	saAux[0] := ('UPDATE `geral`.`processos` SET `InicioAspersao` = $'');
	saAux[1] := (TO_STRING(camara.en.stHoraAgora.wYear));
	saAux[2] := ('-');
	saAux[3] := (TO_STRING(camara.en.stHoraAgora.wMonth));
	saAux[4] := ('-');
	saAux[5] := (TO_STRING(camara.en.stHoraAgora.wDay));
	saAux[6] := (' ');
	saAux[7] := (TO_STRING(camara.en.stHoraAgora.wHour));
	saAux[8] := (':');
	saAux[9] := (TO_STRING(camara.en.stHoraAgora.wMinute));
	saAux[10] := (':');
	saAux[11] := (TO_STRING(camara.en.stHoraAgora.wSecond));
	saAux[12] := ('$' WHERE (`Processo` = $'');
	saAux[13] := (sGuidAnterior);
	saAux[14] := ('$');');
	
	sCmd := F_ConcatArray1000(sArray:= saAux);
	
	aPara.eParaType := E_ExpParameterType.STRING_;
	aPara.nParaSize := SIZEOF(sAux);

	// call functionblock
	IF fbPLCDBaspersao.Execute(
		hDBID:= 1, 
		pExpression:= ADR(sCmd), 
		cbExpression:= SIZEOF(sCmd), 
		pData:= ADR(sAux), 
		cbData:= SIZEOF(sAux), 
		pParameter:= ADR(aPara), 
		cbParameter:= SIZEOF(aPara)) 
	THEN
		IF NOT fbPLCDBaspersao.bError THEN
			xSalvaInicioAspersao := FALSE;
		END_IF
	END_IF
END_IF
END_ACTION

ACTION InicioResfriamento:



//UPDATE `geral`.`processos` SET `InicioResfriamento` = '1', `NumeroCarcacas` = '1' WHERE (`Processo` = '{F4C353B8-2323-45D1-B9F0-8A1F447BE435}');


IF xSalvaResfriamento THEN
	
	FOR i:= 0 TO 50 DO
		saAux[i]:= '';
	END_FOR
	
	saAux[0] := ('UPDATE `geral`.`processos` SET `InicioResfriamento` = $'');
	saAux[2] := (TO_STRING(camara.en.stHoraAgora.wYear));
	saAux[3] := ('-');
	saAux[4] := (TO_STRING(camara.en.stHoraAgora.wMonth));
	saAux[5] := ('-');
	saAux[6] := (TO_STRING(camara.en.stHoraAgora.wDay));
	saAux[7] := (' ');
	saAux[8] := (TO_STRING(camara.en.stHoraAgora.wHour));
	saAux[9] := (':');
	saAux[10] := (TO_STRING(camara.en.stHoraAgora.wMinute));
	saAux[11] := (':');
	saAux[12] := (TO_STRING(stHoraAhora.wSecond));
	saAux[13] := ('$', `NumeroCarcacas` = $'');
	saAux[14] := (TO_STRING(Camara.config.iCarcacasReal));
	saAux[15] := ('$', `Camara` = $'');
	saAux[16] := (TO_STRING(Camara.config.iCamara));
	saAux[17] := ('$' WHERE (`Processo` = $'');
	saAux[18] := (sGuidAnterior);
	saAux[19] := ('$');');
	
	sCmd := F_ConcatArray1000(sArray:= saAux);
	
	aPara.eParaType := E_ExpParameterType.STRING_;
	aPara.nParaSize := SIZEOF(sAux);

	// call functionblock
	IF fbPLCDBResfriamento.Execute(
		hDBID:= 1, 
		pExpression:= ADR(sCmd), 
		cbExpression:= SIZEOF(sCmd), 
		pData:= ADR(sAux), 
		cbData:= SIZEOF(sAux), 
		pParameter:= ADR(aPara), 
		cbParameter:= SIZEOF(aPara)) 
	THEN
		IF NOT fbPLCDBResfriamento.bError THEN
			xSalvaResfriamento := FALSE;
		END_IF
	END_IF
END_IF
END_ACTION

ACTION SalvaGrafico:



//INSERT INTO `geral`.`graficosprocesso` (`Processo`, `rTempTanque`, `rPressaoAnel`, `rUmidadeCamara`, `timestamp`) VALUES ('s', 's', 's', 's', 's');

tonAmostra(IN:= sGuidAtual <> '' AND xAmostra, PT:= T#1M, Q=> , ET=> );
IF tonAmostra.q THEN
	tonAmostra(IN:= FALSE);
	xSalvaGrafico := TRUE;
END_IF


IF xSalvaGrafico THEN
	
	FOR i:= 0 TO 50 DO
		saAux[i]:= '';
	END_FOR
	
	
	saAux[0]:= ('INSERT INTO `geral`.`graficoscamara` (`Processo`, `rUmidadeCamara`, `rTem');
	saAux[1]:= ('peraturaCamara`,`rVazaoCamara`,`rPressaoAnel`,`rTempReservatorio`');
	saAux[2]:= (', `timestamp`) VALUES ($'');
	saAux[3]:= (sGuidAnterior);
	saAux[4]:= ('$', $'');
	saAux[5]:= (TO_STRING(F_RetiraCasa(Entrada:= Camara.en.rUmidadeCamara, casa:=2)));
	saAux[6]:= ('$', $'');
	saAux[7]:= (TO_STRING(F_RetiraCasa(Entrada:= Camara.en.rTempCamara, casa:=2)));
	saAux[8]:= ('$', $'');
	saAux[9]:= (TO_STRING(F_RetiraCasa(Entrada:= Camara.en.rVaozaoInstantanea, casa:=2)));
	saAux[10]:= ('$', $'');
	saAux[11]:= (TO_STRING(F_RetiraCasa(Entrada:= Camara.en.rPressaoAnel, casa:=2)));
	saAux[12]:= ('$', $'');
	saAux[13]:= (TO_STRING(F_RetiraCasa(Entrada:= Camara.en.rTempTanque, casa:=2)));
	saAux[14]:= ('$', $'');
	saAux[15]:= (TO_STRING(camara.en.stHoraAgora.wYear));
	saAux[16]:= ('-');
	saAux[17]:= (TO_STRING(camara.en.stHoraAgora.wMonth));
	saAux[18]:= ('-');
	saAux[19]:= (TO_STRING(camara.en.stHoraAgora.wDay));
	saAux[20]:= (' ');
	saAux[21]:= (TO_STRING(camara.en.stHoraAgora.wHour));
	saAux[22]:= (':');
	saAux[23]:= (TO_STRING(camara.en.stHoraAgora.wMinute));
	saAux[24]:= (':');
	saAux[25]:= (TO_STRING(camara.en.stHoraAgora.wSecond));
	saAux[26]:= ('$');');
	
	sCmd := F_ConcatArray1000(sArray:= saAux);
	
	aPara.eParaType := E_ExpParameterType.STRING_;
	aPara.nParaSize := SIZEOF(sAux);

	// call functionblock
	IF fbPLCDBCmd.Execute(
		hDBID:= 1, 
		pExpression:= ADR(sCmd), 
		cbExpression:= SIZEOF(sCmd), 
		pData:= ADR(sAux), 
		cbData:= SIZEOF(sAux), 
		pParameter:= ADR(aPara), 
		cbParameter:= SIZEOF(aPara)) 
	THEN
		xSalvaGrafico := FALSE;
	END_IF
END_IF
END_ACTION

ACTION SalvaProtocolo:

IF xSalvaProtocolo THEN
		
	FOR i:= 0 TO 50 DO
		saAux[i]:= '';
	END_FOR

	//UPDATE `geral`.`processos` SET `sProtocolo` = 'aaaaaaa' WHERE (`Processo` = '{008089BB-BE64-417E-ABDE-888FE5FB9663}');

	saAux[0] := ('UPDATE `geral`.`processos` SET `sProtocolo` = $'');
	saAux[1] := (Camara.config.stProtocolos[Camara.config.iProtocoloEscolhido].DB.Nome);
	saAux[2] := ('$' WHERE (`Processo` = $'');
	saAux[3] := (sGuidAnterior);
	saAux[4] := ('$');');
	
	sCmd := F_ConcatArray1000(sArray:= saAux);
	
	aPara.eParaType := E_ExpParameterType.STRING_;
	aPara.nParaSize := SIZEOF(sAux);

	// call functionblock
	IF fbPLCDProtocolo.Execute(
		hDBID:= 1, 
		pExpression:= ADR(sCmd), 
		cbExpression:= SIZEOF(sCmd), 
		pData:= ADR(sAux), 
		cbData:= SIZEOF(sAux), 
		pParameter:= ADR(aPara), 
		cbParameter:= SIZEOF(aPara)) 
	THEN
		IF NOT fbPLCDProtocolo.bError THEN
			xSalvaProtocolo := FALSE;
		END_IF
	END_IF
END_IF
END_ACTION

ACTION AjustaEntrada:



IF Camara.config.iCamara <> CamaraAnterior.config.iCamara THEN
	iCamara := Camara.config.iCamara;
END_IF
IF Camara.config.iCamara <> iCamara THEN
	Camara.config.iCamara := iCamara;
END_IF


IF Camara.config.sNome <> CamaraAnterior.config.sNome THEN
	sNome := Camara.config.sNome;
END_IF
IF Camara.config.sNome <> sNome THEN
	Camara.config.sNome := sNome;
END_IF


IF Camara.en.sGuidAtual <> CamaraAnterior.en.sGuidAtual THEN
	sGuidAtual := Camara.en.sGuidAtual;
END_IF
IF Camara.en.sGuidAtual <> sGuidAtual THEN
	Camara.en.sGuidAtual := sGuidAtual;
END_IF


IF Camara.config.sValvulas <> CamaraAnterior.config.sValvulas THEN
	sValvulas := Camara.config.sValvulas;
	F_StringSeparadorFBGrupos(sStr:= sValvulas, ListaINT:=iValvulas);
END_IF
IF Camara.config.sValvulas <> sValvulas THEN
	Camara.config.sValvulas := sValvulas;
	F_StringSeparadorFBGrupos(sStr:= sValvulas, ListaINT:=iValvulas);
END_IF


IF Camara.status.xCamaraTempOK <> CamaraAnterior.status.xCamaraTempOK THEN
	xCamaraTempOK := Camara.status.xCamaraTempOK;
END_IF
IF Camara.status.xCamaraTempOK <> xCamaraTempOK THEN
	Camara.status.xCamaraTempOK := xCamaraTempOK;
END_IF

IF Camara.status.xCamaraUmidOK <> CamaraAnterior.status.xCamaraUmidOK THEN
	xCamaraUmidOK := Camara.status.xCamaraUmidOK;
END_IF
IF Camara.status.xCamaraUmidOK <> xCamaraUmidOK THEN
	Camara.status.xCamaraUmidOK := xCamaraUmidOK;
END_IF

IF Camara.status.xAnelPressOK <> CamaraAnterior.status.xAnelPressOK THEN
	xAnelPressOK := Camara.status.xAnelPressOK;
END_IF
IF Camara.status.xAnelPressOK <> xAnelPressOK THEN
	Camara.status.xAnelPressOK := xAnelPressOK;
END_IF

IF Camara.status.xTanqueTempOK <> CamaraAnterior.status.xTanqueTempOK THEN
	xTanqueTempOK := Camara.status.xTanqueTempOK;
END_IF
IF Camara.status.xTanqueTempOK <> xTanqueTempOK THEN
	Camara.status.xTanqueTempOK := xTanqueTempOK;
END_IF

IF Camara.en.xFinalizaValvulasDaCamara <> CamaraAnterior.en.xFinalizaValvulasDaCamara THEN
	xFinalizaValvulasDaCamara := Camara.en.xFinalizaValvulasDaCamara;
END_IF
IF Camara.en.xFinalizaValvulasDaCamara <> xFinalizaValvulasDaCamara THEN
	Camara.en.xFinalizaValvulasDaCamara := xFinalizaValvulasDaCamara;
END_IF

//Quantidade minima de carcaças a amostrar
IF Camara.config.iCarcacasAmostra < 20 THEN
	Camara.config.iCarcacasAmostra := 20;
END_IF



CamaraAnterior := Camara;
END_ACTION

ACTION AjustaSaida:




Camara.status.sStatus := sStatus;
Camara.status.iStatus := iStatus;
Camara.status.xTerminouAspercao := xTerminouAspercao;
Camara.sa.iQuantidadeDeCluster := iQuantidadeDeCluster;

Camara.status.sNomeProtocoloAtivo := Camara.config.stProtocolos[Camara.sa.iProtocoloAtual].DB.Nome;



Camara.sa.iValvulaMestraMestra := iValvulaMestraMestra;
END_ACTION

ACTION BTPausaECancela:




//Sinal de cancela todas as valvulas
btCancela(CLK:= Camara.en.xCancelaTodas, Q=> );
IF btCancela.q THEN
	xIniciaCascataCancela := TRUE;
END_IF
tonCascataCancela(IN:= xIniciaCascataCancela, PT:= T#250MS, Q=> , ET=> );
IF tonCascataCancela.q THEN
	tonCascataCancela(IN:=FALSE);
	FOR i := 0 TO 500 DO
		IF iValvulas[i] = 0 THEN
			xIniciaCascataCancela := FALSE;
			EXIT;
		ELSE
			//Se esta aspergindo, pausado critico, pausado sinc ou ligado man ele faz de com espaço
			IF stControleValvulas[iValvulas[i]].SA.iStatus <> 9 THEN
				stControleValvulas[iValvulas[i]].EN.xPulaAspersao := TRUE;
				EXIT;//Sai para ter que contar o tempo novamente 
			ELSE
				stControleValvulas[iValvulas[i]].EN.xPulaAspersao := TRUE;
			END_IF
		END_IF
	END_FOR
END_IF







btManualTodas(CLK:= Camara.en.xManualTodas, Q=> );
IF btManualTodas.q THEN
	xManualtodas := Camara.en.xManualTodas;
	IF Camara.en.xManualTodas THEN
		xIniciaInterno := sGuidAtual = '';//Inicia o processo da camara
	ELSE
		xApagaProcessoInterno := true;//quando volta de manual finaliza a camara
	END_IF
	FOR i := 0 TO 500 DO
		IF iValvulas[i] = 0 THEN
			EXIT;
		ELSE
			 stControleValvulas[iValvulas[i]].EN.stValvula.en.xAutomaticoManual := NOT xManualtodas; 
		END_IF
	END_FOR
END_IF






(*
btBTCancelaTudo(CLK:= Camara.en.xBTPausaeCancela, Q=> );
IF btBTCancelaTudo.q THEN
	
	IF xIniciouCancela AND NOT tonBTCancelaTudo.q THEN
		
		xPausaInterno := NOT xPausaInterno;
		FOR i := 0 TO 500 DO
			IF iValvulas[i] = 0 THEN
				EXIT;
			ELSE
				 stControleValvulas[iValvulas[i]].EN.xPausaUsuarioCamara := xPausaInterno; 
			END_IF
		END_FOR
		Camara.sa.xLedBTPausaeCancela := xPausaInterno;
	
	END_IF
	
	xIniciouCancela := Camara.en.xBTPausaeCancela;
END_IF



//Se segura o botao por mais de x tempo ele passa cancelando todas as valvulas
tonBTCancelaTudo(IN:= Camara.en.xBTPausaeCancela, PT:= T#5S, Q=> , ET=> );
rtCancelaInterno(CLK:= tonBTCancelaTudo.q, Q=> );
IF rtCancelaInterno.q THEN
	FOR i := 0 TO 500 DO
		IF iValvulas[i] = 0 THEN
			EXIT;
		ELSE
			 stControleValvulas[iValvulas[i]].EN.xPulaAspersao := TRUE; 
		END_IF
	END_FOR
END_IF



//Se segurar apertado vai apagar o processo todo
tonBTCancelaTudoApagaProcesso(IN:= Camara.en.xBTPausaeCancela, PT:=T#10S , Q=> , ET=> );
rtBTCancelaTudoApagaProcesso(CLK:= tonBTCancelaTudoApagaProcesso.q, Q=> );
IF rtBTCancelaTudoApagaProcesso.q THEN
	Camara.en.xApagaProcessoSupervisorio := TRUE;
END_IF
*)
END_ACTION

ACTION ConsumoAgua:




CASE Camara.Config.iTipoMedicaoAgua OF
	
	0://Por fora
	
	
	
	1://Hidrometro
	
		fbHibrometro(	rContador:= Camara.Retentivas.rHidrometroTotal, 
						rContadorHoje:= Camara.Retentivas.rHidrometroHoje, 
						Historico:= Camara.Retentivas.HistoricoHidrometro, 
						xSinal:= Camara.en.xSensorVazao, 
						xResetContador:= , 
						rMultiplicadorVazao:= Camara.Config.rMultiplicadorVazao, 
						stHoraAgora:= stHoraAhora);
	
	
	
	2://Vazao instantanea
	
		fbTotalizadorVazao(	HistoricoHidrometro:= Camara.Retentivas.HistoricoHidrometro, 
							rVazaoTotalHoje:= Camara.Retentivas.rHidrometroHoje, 
							rVazaoTotalHistorica:= Camara.Retentivas.rHidrometroTotal, 
							stHoraAgora:= stHoraAhora, 
							rVazaoInstantanea:= Camara.en.rVaozaoInstantanea);
	
	
	
END_CASE
END_ACTION

ACTION ControleLed:


ton10s(IN:=TRUE, PT:= T#10S, Q=> , ET=> );
IF ton10s.q THEN
	ton10s(IN:=false);
	x10s := NOT x10s;
END_IF

ton2s(IN:=TRUE, PT:= T#2S, Q=> , ET=> );
IF ton2s.q THEN
	ton2s(IN:=FALSE);
	x2s := NOT x2s;
END_IF

ton500ms(IN:=TRUE, PT:= T#500MS, Q=> , ET=> );
IF ton500ms.q THEN
	ton500ms(IN:=FALSE);
	x500ms := NOT x500ms;
END_IF


IF sGuidAtual = '' THEN
	Camara.sa.xLed := FALSE;	
END_IF

IF sGuidAtual <> '' AND NOT xIniciouAspercao THEN
	Camara.sa.xLed := x2s;
END_IF

IF sGuidAtual <> '' AND xIniciouAspercao THEN
	Camara.sa.xLed := TRUE;
END_IF

IF sGuidAtual <> '' AND xTerminouAspercao THEN
	Camara.sa.xLed := x10s AND x2s;
END_IF



IF Camara.en.xLedManual THEN
	Camara.sa.xLed := Camara.en.xSinalManuLed;
END_IF
END_ACTION

ACTION InicioPelaCamara:



CASE iMaquinaIniciaSemPeso OF
	0://Esperando ter que criar um guid e salvar no banco
		IF (Camara.en.xIniciaCamaraSupervisorio OR Camara.en.xIniciaCamaraIHM OR xIniciaInterno) AND sGuidAtual = '' THEN
			iMaquinaIniciaSemPeso := 1;
			Camara.en.xIniciaCamaraSupervisorio := FALSE;
			Camara.en.xIniciaCamaraIHM := FALSE;
			xIniciaInterno := false;
		END_IF
		
	1: // cria o guid
	
		fbCriaGUID(
			bExecute:= TRUE,  
			sNetId:= '', 
			tTimeout:= T#5S, 
			pGuidBuffer:= ADR(guidCriado), 
			nGuidBufferSize:= SIZEOF(guidCriado), 
			bBusy=> , 
			bError=> , 
			nErrorId=> );
			
		IF NOT fbCriaGUID.bBusy THEN
			fbCriaGUID(bExecute:= FALSE);
			sGuidAtual := GUID_TO_REGSTRING(guidCriado);
			iMaquinaIniciaSemPeso := 2;
		END_IF
		
	2://salva no banco o role
		FOR i:= 0 TO 50 DO
			saAux[i]:= '';
		END_FOR
	
		saAux[0] := ('INSERT INTO `geral`.`processos` (`Processo`');
		saAux[1] := (', `Camara`, `Status`,`InicioResfriamento`, `Timestamp`) VALUES ($'');
		saAux[2] := sGuidAtual;
		saAux[3] := '$', $'';
		saAux[4] := TO_STRING(Camara.config.iCamara);
		saAux[5] := '$', $'';
		saAux[6] := 'Esperando aspersao';
		saAux[7] := '$', $'';
		saAux[8] := TO_STRING(stHoraAhora.wYear);
		saAux[9] := ('-');
		saAux[10] := (TO_STRING(stHoraAhora.wMonth));
		saAux[11] := ('-');
		saAux[12] := (TO_STRING(stHoraAhora.wDay));
		saAux[13] := (' ');
		saAux[14] := (TO_STRING(stHoraAhora.wHour));
		saAux[15] := (':');
		saAux[16] := (TO_STRING(stHoraAhora.wMinute));
		saAux[17] := (':');
		saAux[18] := (TO_STRING(stHoraAhora.wSecond));
		saAux[19] := '$', $'';
		saAux[20] := TO_STRING(stHoraAhora.wYear);
		saAux[21] := ('-');
		saAux[22] := (TO_STRING(stHoraAhora.wMonth));
		saAux[23] := ('-');
		saAux[24] := (TO_STRING(stHoraAhora.wDay));
		saAux[25] := (' ');
		saAux[26] := (TO_STRING(stHoraAhora.wHour));
		saAux[27] := (':');
		saAux[28] := (TO_STRING(stHoraAhora.wMinute));
		saAux[29] := (':');
		saAux[30] := (TO_STRING(stHoraAhora.wSecond));
		saAux[31] := ('$');');
		
		sCmd := F_ConcatArray1000(sArray:= saAux);
		
		aPara.eParaType := E_ExpParameterType.STRING_;
		aPara.nParaSize := SIZEOF(sAux);
	
		// call functionblock
		IF fbDBInicioProcesso.Execute(
			hDBID:= 1, 
			pExpression:= ADR(sCmd), 
			cbExpression:= SIZEOF(sCmd), 
			pData:= ADR(sAux), 
			cbData:= SIZEOF(sAux), 
			pParameter:= ADR(aPara), 
			cbParameter:= SIZEOF(aPara)) 
		THEN
			IF NOT fbDBInicioProcesso.bError THEN
				xSalvaIniSemPeso := TRUE;
				iMaquinaIniciaSemPeso := 0;
			END_IF
		END_IF
END_CASE
END_ACTION

ACTION Status:

(*status
1 = cinza = StandBy
2 = amarelo = Aguardando inicio (Pos pesagem quente)
3 = azul escuro = Aspergindo automatico
4 = preto = Finalizada
5 = Vermelho = Pausado
6 = Laranja = Cancelado
7 = Roxo = Manual
8 = Verde = Coletando pesoso quentes
9 = Azul claro = Coletando pesoso frios
*)


IF sGuidAtual = '' THEN
	
	CASE Camara.Config.Linguagem OF
		enu_Linguagem.Portugues:
			sStatus := 'StandBy';
		enu_Linguagem.Espanhol:
			sStatus := 'StandBy';
		enu_Linguagem.Ingles:
			sStatus := 'StandBy';
	END_CASE
	
	iStatus := 1;
ELSE
	
	//Se nenhum vai para standby
	CASE Camara.Config.Linguagem OF
		enu_Linguagem.Portugues:
			sStatus := 'StandBy';
		enu_Linguagem.Espanhol:
			sStatus := 'StandBy';
		enu_Linguagem.Ingles:
			sStatus := 'StandBy';
	END_CASE
	
	iStatus := 1;


	
	IF Camara.Status.xPegandoPesosQuentes THEN
		CASE Camara.Config.Linguagem OF
			enu_Linguagem.Portugues:
				sStatus := 'Aquisitando pesos quentes';
			enu_Linguagem.Espanhol:
				sStatus := 'Adquisición de pesos calientes';
			enu_Linguagem.Ingles:
				sStatus := 'Acquiring hot weights';
		END_CASE
		iStatus := 8;
	END_IF
	(*
	IF NOT xIniciouAspercao AND NOT Camara.Status.xPegandoPesosQuentes THEN
		CASE Camara.Config.Linguagem OF
			enu_Linguagem.Portugues:
				sStatus := 'Esperando o incio da aspersão';
			enu_Linguagem.Espanhol:
				sStatus := 'Esperando a que arranque el aspersor';
			enu_Linguagem.Ingles:
				sStatus := 'Waiting for the sprinkler to start';
		END_CASE
		iStatus := 2;
	END_IF*)
	
	IF NOT xTerminouAspercao AND xIniciouAspercao THEN
		CASE Camara.Config.Linguagem OF
			enu_Linguagem.Portugues:
				sStatus := 'Esperando o fim da aspersão';
			enu_Linguagem.Espanhol:
				sStatus := 'Esperando el final de la aspersión';
			enu_Linguagem.Ingles:
				sStatus := 'Waiting for the end of the sprinkling';
		END_CASE
		iStatus := 3;
	END_IF
	
	IF xTerminouAspercao THEN
		CASE Camara.Config.Linguagem OF
			enu_Linguagem.Portugues:
				sStatus := 'Aspersão finalizada';
			enu_Linguagem.Espanhol:
				sStatus := 'Aspersión finalizado';
			enu_Linguagem.Ingles:
				sStatus := 'Sprinkling finished';
		END_CASE
		iStatus	 := 4;
	END_IF
	
	
	IF Camara.Status.xPegandoPesosFrios THEN
		CASE Camara.Config.Linguagem OF
			enu_Linguagem.Portugues:
				sStatus := 'Aquisitando pesos frios';
			enu_Linguagem.Espanhol:
				sStatus := 'Adquirir pesos en frío';
			enu_Linguagem.Ingles:
				sStatus := 'Acquiring cold weights';
		END_CASE
		iStatus := 9;
	END_IF
	
	//Abaixo os prioritarios sobre esses de cima
	
	IF Camara.Status.xPeloMenos1CanceladaOutrasAguradando OR Camara.Status.xTodasValvulasCanceladas THEN
		iStatus	 := 6;
	END_IF
	
	IF Camara.Status.xAlgumaValvulaEmManual THEN
		iStatus	 := 7;
	END_IF
	
	IF Camara.en.xPausaUsuario THEN
		CASE Camara.Config.Linguagem OF
			enu_Linguagem.Portugues:
				sStatus := 'Pausa pelo usuario';
			enu_Linguagem.Espanhol:
				sStatus := 'Pausa por el usuario';
			enu_Linguagem.Ingles:
				sStatus := 'Pausa pelo usuario';
		END_CASE
		iStatus	 := 2;
	END_IF
	
	
	
	IF (NOT xCamaraTempOK OR NOT xCamaraUmidOK OR NOT xAnelPressOK OR NOT xTanqueTempOK OR NOT Camara.en.xEmergenciaOK) AND NOT xTerminouAspercao THEN	
		iStatus	 := 5;		
	END_IF
END_IF



//Tem alguma Valvula em manual
Camara.Status.xAlgumaValvulaEmManual := FALSE;
FOR i := 0 TO 500 DO
	IF iValvulas[i] = 0 THEN
		EXIT;
	ELSE
		IF NOT stControleValvulas[iValvulas[i]].EN.stValvula.en.xAutomaticoManual THEN
			Camara.Status.xAlgumaValvulaEmManual := TRUE;	
		END_IF
	END_IF
END_FOR



//Ve se tem pelo menos 1 valvula cancelada e as outras estao aguardando
//Bah o nome ficou errado aqui :( e agora nao da pra alterar
//Se tu ver isso mais tarde ajusta o nome aqui pra nao ficar xTodasValvulasCanceladas
Camara.Status.xPeloMenos1CanceladaOutrasAguradando := FALSE;	
FOR i := 0 TO 500 DO
	IF iValvulas[i] = 0 THEN
		EXIT;
	ELSE
		//Se tiver 
		IF stControleValvulas[iValvulas[i]].SA.iStatus = 9 THEN
			Camara.Status.xPeloMenos1CanceladaOutrasAguradando := TRUE;	
			EXIT;
		END_IF
	END_IF
END_FOR
FOR i := 0 TO 500 DO
	IF iValvulas[i] = 0 THEN
		EXIT;
	ELSE
		//Se tiver 
		IF stControleValvulas[iValvulas[i]].SA.iStatus <> 9 AND stControleValvulas[iValvulas[i]].SA.iStatus <> 4 THEN
			Camara.Status.xPeloMenos1CanceladaOutrasAguradando := FALSE;	
			EXIT;
		END_IF
	END_IF
END_FOR



Camara.Status.xTodasValvulasCanceladas := TRUE;
FOR i := 0 TO 500 DO
	IF iValvulas[i] = 0 THEN
		EXIT;
	ELSE
		//Se tiver 
		IF stControleValvulas[iValvulas[i]].SA.iStatus <> 9 THEN
			Camara.Status.xTodasValvulasCanceladas := FALSE;		
			EXIT;
		END_IF
	END_IF
END_FOR



//Tudas Pausadas Pelo Usuario 
Camara.Status.xTudoPausadoPeloUsuario := TRUE;
FOR i := 0 TO 500 DO
	IF iValvulas[i] = 0 THEN
		EXIT;
	ELSE
		IF NOT stControleValvulas[iValvulas[i]].EN.xPausaUsuarioCamara THEN
			Camara.Status.xTudoPausadoPeloUsuario := FALSE;		
			EXIT;
		END_IF
	END_IF
END_FOR

Camara.Status.xTudoPausadoPeloUsuario := Camara.en.xPausaUsuario;


//Pelo menos 1 finalizada as outras canceladas
Camara.Status.xPeloMenos1FinalizadaOutrasCanceladas := FALSE;	
FOR i := 0 TO 500 DO
	IF iValvulas[i] = 0 THEN
		EXIT;
	ELSE
		//Se tiver 
		IF stControleValvulas[iValvulas[i]].SA.iStatus = 3 THEN
			Camara.Status.xPeloMenos1FinalizadaOutrasCanceladas := TRUE;	
			EXIT;
		END_IF
	END_IF
END_FOR
FOR i := 0 TO 500 DO
	IF iValvulas[i] = 0 THEN
		EXIT;
	ELSE
		//Se tiver 
		IF stControleValvulas[iValvulas[i]].SA.iStatus <> 9 AND stControleValvulas[iValvulas[i]].SA.iStatus <> 3 THEN
			Camara.Status.xPeloMenos1FinalizadaOutrasCanceladas := FALSE;	
			EXIT;
		END_IF
	END_IF
END_FOR




Camara.en.xHabilitaAtualizarCluster := sGuidAtual = '' OR (iStatus = 4 OR iStatus = 1 OR iStatus = 2);
IF sGuidAtual <> '' THEN
	Camara.sa.tHoraTermina := DT#1970-01-01-00:00;
	FOR i := 0 TO 500 DO
		IF iValvulas[i] = 0 THEN
			EXIT;
		ELSE
			//COntrole de que hora termina
			IF stControleValvulas[iValvulas[i]].SA.dtHoraTermina > Camara.sa.tHoraTermina THEN
				Camara.sa.tHoraTermina := stControleValvulas[iValvulas[i]].SA.dtHoraTermina;
			END_IF
			
			//COntrole se pode trocar o protocolo e se pode editar os clisters
			IF stControleValvulas[iValvulas[i]].SA.xEmProcesso AND NOT stControleValvulas[iValvulas[i]].SA.iStatus = 3 AND NOT stControleValvulas[iValvulas[i]].SA.iStatus = 9 THEN
				//Camara.xHabilitaAtualizarCluster := FALSE;
			END_IF
		END_IF
	END_FOR
END_IF


Camara.sa.sHoraTermina := REPLACE(STR1:= TO_STRING(Camara.sa.tHoraTermina), STR2:= '', L:= 15, P:=0);
Camara.sa.sHoraInicio := REPLACE(STR1:= TO_STRING(Camara.sa.tHoraInicio), STR2:= '', L:= 15, P:=0);
END_ACTION

ACTION StatusLedVermelhoDoGaja:

//programa feito com muito amor para o led vermelho do gaja (Aspersao de rosario, mais uma vez patrocinada pela eng da metal marc, o pessoal que sabe fazer projeto)






Camara.Status.iStatusBotaoVermelho := 0;

IF Camara.Status.xTodasValvulasCanceladas THEN
	Camara.Status.iStatusBotaoVermelho := 1;
END_IF

IF Camara.Status.xTudoPausadoPeloUsuario THEN
	Camara.Status.iStatusBotaoVermelho := 2;
END_IF

IF Camara.Status.xPeloMenos1FinalizadaOutrasCanceladas THEN
	Camara.Status.iStatusBotaoVermelho := 3;
END_IF
END_ACTION

END_FUNCTION_BLOCK

// POUs/Automatico/Aspercao/Camaras/FB_SalvaEventoRelatorio
FUNCTION_BLOCK FB_SalvaEventoRelatorio
VAR_INPUT
	sGuid : STRING;
	xInicio : BOOL;
	xCritico : BOOL;
	sDescricao : STRING;
	sTag : STRING;
	iCamara : INT;
	stHoraAgora : TIMESTRUCT;
END_VAR
VAR_OUTPUT
END_VAR
VAR
	stEvento : st_EventoRelatorio;
	rtComecou : R_TRIG;
	ftTerminou : f_TRIG;
	xSalva : BOOL;
	saAux : ARRAY[0..50] OF STRING(80);
	i : INT;
	
	fbPLCDBCmd    : FB_PLCDBCmdEvt(sNetID := '', tTimeout := T#5S);
    sCmd          : STRING (1000); 
    aPara         : ST_ExpParameter;
	sAux 		  : STRING;
END_VAR



IF xLicensaValida6446896834 THEN	

	rtComecou(CLK:= xInicio, Q=> );
	IF rtComecou.q THEN
		stEvento.Inicio := stHoraAgora;
	END_IF
	
	ftTerminou(CLK:= xInicio, Q=> );
	IF ftTerminou.q THEN
		stEvento.Fim := stHoraAgora;
		xSalva := TRUE;
	END_IF
	
	
	stEvento.sGuid := sGuid;
	stEvento.Critico := xCritico;
	stEvento.Descricao := sDescricao;
	stEvento.Tag := sTag;
	stEvento.iCamara := iCamara;
	
	
	SalvaEvento();
	

ELSE
	
	ValidaLicensa();

END_IF

ACTION SalvaEvento:



//INSERT INTO `geral`.`eventosreltaorio` (`Processo`, `iCamara`, `Critico`, `Tag`, `Descricao`, `Inicio`, `Fim`, `Timestamp`) VALUES ('{F0DC1A48-C5E7-44DB-AEEC-A20D89C0E82A}', '44', '1', 'PressaoAnel', 'Pressão no anel inferior 0.5 bar', '2023-12-11 11:21:27', '2023-12-11 12:07:12', '2023-12-11 12:07:12');


IF xSalva THEN
	
	FOR i:= 0 TO 50 DO
		saAux[i] := '';
	END_FOR

	saAux[0] := 'INSERT INTO `geral`.`eventosreltaorio` (`Processo`, `iCamara`,';
	saAux[1] := ' `Critico`, `Tag`, `Descricao`, `Inicio`, `Fim`, `Timestamp`) VALUES ($'';
	saAux[2] := (stEvento.sGuid);
	saAux[3] := ('$', $'');
	saAux[4] := (TO_STRING(stEvento.iCamara));
	saAux[5] := ('$', $'');
	IF stEvento.Critico THEN
		saAux[6] := (TO_STRING(1));
	ELSE
		saAux[6] := (TO_STRING(0));
	END_IF
	saAux[7] := ('$', $'');
	saAux[8] := ((stEvento.Tag));
	saAux[9] := ('$', $'');
	saAux[10] := ((stEvento.Descricao));
	saAux[11] := ('$', $'');
	saAux[12] := (TO_STRING(stEvento.Inicio.wYear));
	saAux[13] := ('-');
	saAux[14] := (TO_STRING(stEvento.Inicio.wMonth));
	saAux[15] := ('-');
	saAux[16] := (TO_STRING(stEvento.Inicio.wDay));
	saAux[17] := (' ');
	saAux[18] := (TO_STRING(stEvento.Inicio.wHour));
	saAux[19] := (':');
	saAux[20] := (TO_STRING(stEvento.Inicio.wMinute));
	saAux[21] := (':');
	saAux[22] := (TO_STRING(stEvento.Inicio.wSecond));
	saAux[23] := ('$', $'');
	saAux[24] := (TO_STRING(stEvento.fim.wYear));
	saAux[25] := ('-');
	saAux[26] := (TO_STRING(stEvento.fim.wMonth));
	saAux[27] := ('-');
	saAux[28] := (TO_STRING(stEvento.fim.wDay));
	saAux[29] := (' ');
	saAux[30] := (TO_STRING(stEvento.fim.wHour));
	saAux[31] := (':');
	saAux[32] := (TO_STRING(stEvento.fim.wMinute));
	saAux[33] := (':');
	saAux[34] := (TO_STRING(stEvento.fim.wSecond));
	saAux[35] := ('$', $'');
	saAux[36] := (TO_STRING(stHoraAgora.wYear));
	saAux[37] := ('-');
	saAux[38] := (TO_STRING(stHoraAgora.wMonth));
	saAux[39] := ('-');
	saAux[40] := (TO_STRING(stHoraAgora.wDay));
	saAux[41] := (' ');
	saAux[42] := (TO_STRING(stHoraAgora.wHour));
	saAux[43] := (':');
	saAux[44] := (TO_STRING(stHoraAgora.wMinute));
	saAux[45] := (':');
	saAux[46] := (TO_STRING(stHoraAgora.wSecond));
	saAux[47] := ('$');');
	
	
	
	sCmd := F_ConcatArray1000(sArray:= saAux);
	
	
	
	aPara.eParaType := E_ExpParameterType.STRING_;
	aPara.nParaSize := SIZEOF(sAux);

	// call functionblock
	IF fbPLCDBCmd.Execute(
		hDBID:= 1, 
		pExpression:= ADR(sCmd), 
		cbExpression:= SIZEOF(sCmd), 
		pData:= ADR(sAux), 
		cbData:= SIZEOF(sAux), 
		pParameter:= ADR(aPara), 
		cbParameter:= SIZEOF(aPara)) 
	THEN
		xSalva := FALSE;
	END_IF
END_IF
END_ACTION

END_FUNCTION_BLOCK

// POUs/Automatico/Aspercao/ControleLiberacaoCamaras/AreaFria/FB_ControleSaidaAreaFria
FUNCTION_BLOCK FB_ControleSaidaAreaFria
VAR_IN_OUT
	stFria : st_AreaFria;
	stCamaras : ARRAY[*] OF st_Camara;
END_VAR
VAR_INPUT
	iCamaraSelecionada	: INT;// qual camara o operador escolher para começar
	xIniciaCamara		: BOOL;// operador dizendo para começar a amostragem
	xAleatorio			: BOOL;// se vai fazer a amostragem aleatorio ou sequencial
	xCapturaPeso		: BOOL;// operador dizendo para pegar o peso atual
	rPesoAtual			: REAL;// Peso atual que vem da balança
	xPesoNovo			: BOOL;// Quando  balança diz que veio um peso novo
	stHoraAhora 		: TIMESTRUCT; //Hora atual 
END_VAR
VAR_OUTPUT	
	iCamarasDisponiveis : ARRAY[0..50] OF INT; // para a lista do cara para escolher a camara
	rPesosFrios			: ARRAY[0..1000] OF REAL; // 	array com os frios quentes amostrados pelo operador ou sequencialmente
	rPesosQuentes		: ARRAY[0..1000] OF REAL; // 	array com os pesos quentes amostrados pelo operador ou sequencialmente
	sGuidAtual			: STRING;// guid do processo atual
	iCarcacaAtual		: INT;// Qual o numero da carcaça que ele ta esperando
	xPesoOK				: BOOL; //Variavel de controle se o peso esta ok apos as mediçoes
	iNumeroAmostras		: INT;
	xEmProcesso 		: BOOL;
END_VAR
VAR
	stFriaAnterior : st_AreaFria;
	
	iMinCamaras : DINT;
	iMaxCamaras : DINT;
	iAux : INT;
	i : INT;
	iEstado : INT;

	rPesoFrioTotal : REAL;
	rPesoQuenteTotal : REAL;
	xCamaraSelecionadaOK : BOOL;
	xGravaPesoFrio : BOOL;
	xGravaTotalFrio : BOOL;
	
	sSBResfriamentoaaa 	: FB_StringBuilder;
	sSBaaa		  		: FB_StringBuilder;
	fbSBaaa				: FB_StringBuilder;
    fbPLCDBCmd,fbPLCDIgnoraCarcaca 	: FB_PLCDBCmdEvt(sNetID := '', tTimeout := T#2S);
    fbPLCDBRefrimaentoCmd    : FB_PLCDBCmdEvt(sNetID := '', tTimeout := T#2S);
    sCmd          : STRING (1000); 
    aPara         : ST_ExpParameter;
	sAux 		  : STRING;
	saAux 		  : ARRAY[0..50] OF STRING(255);
	xGravaPesoFrioProcesso : BOOL;
	
	
	diAux : DINT;
	
	
	fbProcessoEmail : NT_StartProcess;
	sComando: STRING;
	xGeraRelatorio : BOOL;
	
	rtNovoPeso : R_TRIG;
	xTeste : BOOL;
	xSalvaResfriamento : BOOL;
	
	j : INT := 1;
	
	rPesoSalvar : REAL;
	
	xCacacasIgnoradas : ARRAY[1..20] OF BOOL;
	rtCacacasAIgnorar : ARRAY[1..20] OF R_TRIG;
	
	
	fbSalvaEvento : ARRAY[0..5] OF FB_SalvaEventoRelatorio;
	xSalvaIgnoraCarcaca : BOOL;
	iCarcacaIgnorada : INT;
	
	rtCarcacaIgnorada : R_TRIG;

END_VAR

IF TRUE THEN

	AjustaEntrada();
	PegaCamarasDisponiveis();
	
	
	
	
	
	CASE iEstado OF
		0://Esperando
		//fazer esquema pra ver se a camara selecionada esta dentro das que da pra selecionar
			xCamaraSelecionadaOK := FALSE;
			FOR i := 0 TO 50 DO
				IF iCamarasDisponiveis[i] = 0 THEN
					//EXIT;
				ELSE
					xCamaraSelecionadaOK := xCamaraSelecionadaOK OR iCamaraSelecionada = iCamarasDisponiveis[i];
				END_IF
			END_FOR
			
			xEmProcesso := FALSE;
			
			IF xCamaraSelecionadaOK AND (xIniciaCamara OR stFria.Sup.xIniciarAmostragem OR stFria.IHM.EN.xIniciaAmostragemSequencialTX) THEN
				iEstado := 1;
				rPesosQuentes := stCamaras[iCamaraSelecionada].en.rPesosQuente;
				sGuidAtual 	:= stCamaras[iCamaraSelecionada].en.sGuidAtual;
				stCamaras[iCamaraSelecionada].Status.xPegandoPesosFrios := TRUE;
				iNumeroAmostras := stCamaras[iCamaraSelecionada].config.iCarcacasAmostra;
				
				xIniciaCamara := FALSE;
				iCarcacaAtual := 1;
				stFria.c.xEmProcesso := TRUE;
				xSalvaResfriamento := TRUE;
				
				FOR i := 1 TO 20 DO
					xCacacasIgnoradas[i] := FALSE;
					rtCacacasAIgnorar[i](CLK := FALSE);
				END_FOR
			END_IF
		
		1://Aquisita o peso frio das carcaças e salva no banco
		
			xEmProcesso := TRUE;
		
			IF iCarcacaAtual > iNumeroAmostras AND NOT xIniciaCamara  THEN
				iEstado := 3;
				xGravaPesoFrioProcesso := TRUE;
			END_IF
			
			
			VeCarcacasAIgnorar();
			
			
			rtNovoPeso(CLK:= xPesoNovo OR xTeste OR stFria.Sup.xNovoPesoDebug, Q=> );
			IF rtNovoPeso.q THEN
				IF stFria.Sup.xNovoPesoDebug THEN
					rPesoAtual := stFria.Sup.rPesoDebug;
				END_IF
			END_IF
			
			IF //((xAleatorio AND xCapturaPeso) OR//Se for quando o operador amortrar
			   (NOT xAleatorio AND rtNovoPeso.q) AND//Se for sequencial
				rPesoAtual > 10 THEN // so garante que o peso nao é zero nem muito baixo
			   
				//Se a carcaça foi ignorada, zera ela pro somatorio. e joga o peso dessa carcaca pra proxima
				IF xCacacasIgnoradas[iCarcacaAtual] THEN
					rPesosFrios[iCarcacaAtual] := 0;
					rPesosQuentes[iCarcacaAtual] := 0;
					
					
					//Procura a proxima que ta livre
					FOR i := iCarcacaAtual TO 20 DO
						IF NOT xCacacasIgnoradas[i] THEN
							iCarcacaAtual := i;
							EXIT;
						END_IF
					END_FOR
					
				END_IF
				
				rPesosFrios[iCarcacaAtual] := rPesoAtual;
				rPesoSalvar := rPesoAtual;
				iEstado := 2;
				xGravaPesoFrio := TRUE;
				xPesoNovo := FALSE;
				xCapturaPeso := FALSE;
			END_IF
			
		
		2://Ajusta peso no banco
		
			EscrevePesoFrioCarcaca();
			
			IF NOT xGravaPesoFrio THEN
				iCarcacaAtual := iCarcacaAtual + 1;
				iEstado := 1;
			END_IF
			
			xEmProcesso := TRUE;
			
			
		3://Ve se deu pra cima e salva no banco
		
			xEmProcesso := TRUE;
			rPesoFrioTotal := 0;
			rPesoQuenteTotal := 0;
			
			FOR i := 1 TO 1000 DO
				IF rPesosFrios[i] = 0 AND rPesosQuentes[i] = 0  THEN
					EXIT;
				END_IF
				rPesoFrioTotal := rPesoFrioTotal + rPesosFrios[i];
				rPesoQuenteTotal := rPesoQuenteTotal + rPesosQuentes[i];
			END_FOR
			
			xPesoOK := rPesoQuenteTotal >= rPesoFrioTotal;
			
			EscrevePesoFrioProcesso();
			
			IF NOT xGravaPesoFrioProcesso THEN
				IF xPesoOK THEN
					iEstado := 4;//Deu boa os pesos
				ELSE
					iEstado := 4;//Deu ruim os pesos, ajuste tecnico
				END_IF
			END_IF
			
			
		4://Peso ok ele tira o guid da camara marca como finalizado
			xEmProcesso := TRUE;
			//Zera a camara
			stCamaras[iCamaraSelecionada].en.sGuidAtual := '';
			stCamaras[iCamaraSelecionada].Status.xPegandoPesosFrios := FALSE;
			FOR i := 1 TO 1000 DO
				rPesosFrios[i] := 0;
				rPesosQuentes[i] := 0;
			END_FOR
			sGuidAtual := '';
			stFria.c.xEmProcesso := FALSE;
			iCarcacaAtual := 1;
			iCamaraSelecionada := 0;
			iEstado := 0;//Deu boa os pesos
		
		5://QUando da ruim nos pesos, teria que fazer a repesagem
		
		
	END_CASE
	
	
	FimRefrimento();
	
	SalvaEvento();
	DefineQuandoSalvaEvento();
	IgnoraCarcacaBanco();
	
	
	
	AjustaSaida();
	
	i := j;
	
	
	


END_IF

ACTION DefineQuandoSalvaEvento:




//Carcaca ignorada
rtCarcacaIgnorada(CLK:= xSalvaIgnoraCarcaca, Q=> );
IF rtCarcacaIgnorada.q THEN
	fbSalvaEvento[0].xInicio := TRUE;
	fbSalvaEvento[0].sDescricao := CONCAT('A carcaça N',CONCAT(TO_STRING(iCarcacaIgnorada),' foi ignorada.'));
ELSE
	fbSalvaEvento[0].xInicio := FALSE;
END_IF
END_ACTION

ACTION EscrevePesoFrioCarcaca:


		
IF xGravaPesoFrio THEN
	

	sGuidAtual 	:= stCamaras[iCamaraSelecionada].en.sGuidAtual;
	
	sSBaaa.Clear();
	sSBaaa.Append('UPDATE Carcaca SET PesoFrio = $'');
	sSBaaa.Append(TO_STRING(rPesoSalvar));
	sSBaaa.Append('$', `horaPesoFrio` = $'');
	sSBaaa.Append(TO_STRING(stHoraAhora.wYear));
	sSBaaa.Append('-');
	sSBaaa.Append(TO_STRING(stHoraAhora.wMonth));
	sSBaaa.Append('-');
	sSBaaa.Append(TO_STRING(stHoraAhora.wDay));
	sSBaaa.Append(' ');
	sSBaaa.Append(TO_STRING(stHoraAhora.wHour));
	sSBaaa.Append(':');
	sSBaaa.Append(TO_STRING(stHoraAhora.wMinute));
	sSBaaa.Append(':');
	sSBaaa.Append(TO_STRING(stHoraAhora.wSecond));
	sSBaaa.Append('$' WHERE Processo = $'');
	sSBaaa.Append(sGuidAtual);
	sSBaaa.Append('$' and nCarcaca = $'');
	sSBaaa.Append(TO_STRING(iCarcacaAtual));
	sSBaaa.Append('$';');
	
	sCmd := sSBaaa.GetString();
	
	aPara.eParaType := E_ExpParameterType.STRING_;
	aPara.nParaSize := SIZEOF(sAux);

	// call functionblock
	IF fbPLCDBCmd.Execute(
		hDBID:= 1, 
		pExpression:= ADR(sCmd), 
		cbExpression:= SIZEOF(sCmd), 
		pData:= ADR(sAux), 
		cbData:= SIZEOF(sAux), 
		pParameter:= ADR(aPara), 
		cbParameter:= SIZEOF(aPara)) 
	THEN	
		IF NOT fbPLCDBCmd.bError THEN
			xGravaPesoFrio := FALSE;
		END_IF
	END_IF
END_IF
END_ACTION

ACTION EscrevePesoFrioProcesso:


		
IF xGravaPesoFrioProcesso THEN
	
	sSBaaa.Clear();
	sSBaaa.Append('UPDATE `geral`.`processos` SET `Pesofrio` = $'');
	sSBaaa.Append(TO_STRING(rPesoFrioTotal));
	IF NOT xPesoOK THEN
		sSBaaa.Append('$', `Status` = $'Peso acima');
	ELSE
		sSBaaa.Append('$', `Status` = $'Peso OK');
		sSBaaa.Append('$', `Finalizado` = $'1');
	END_IF
	sSBaaa.Append('$' WHERE (`Processo` = $'');
	sSBaaa.Append(sGuidAtual);
	sSBaaa.Append('$');');
	
	sCmd := sSBaaa.GetString();
	
	aPara.eParaType := E_ExpParameterType.STRING_;
	aPara.nParaSize := SIZEOF(sAux);

	// call functionblock
	IF fbPLCDBCmd.Execute(
		hDBID:= 1, 
		pExpression:= ADR(sCmd), 
		cbExpression:= SIZEOF(sCmd), 
		pData:= ADR(sAux), 
		cbData:= SIZEOF(sAux), 
		pParameter:= ADR(aPara), 
		cbParameter:= SIZEOF(aPara)) 
	THEN	
		IF NOT fbPLCDBCmd.bError THEN
			xGravaPesoFrioProcesso := FALSE;
			xGeraRelatorio := true;
		END_IF
	END_IF
END_IF
END_ACTION

ACTION FimRefrimento:



//UPDATE `geral`.`processos` SET `FimResfriamento` = '2020-12-02 15:00:00' WHERE (`Processo` = 'teste');


IF xSalvaResfriamento THEN
	sSBResfriamentoaaa.Clear();
	sSBResfriamentoaaa.Append('UPDATE `geral`.`processos` SET `FimResfriamento` = $'');
	sSBResfriamentoaaa.Append(TO_STRING(stHoraAhora.wYear));
	sSBResfriamentoaaa.Append('-');
	sSBResfriamentoaaa.Append(TO_STRING(stHoraAhora.wMonth));
	sSBResfriamentoaaa.Append('-');
	sSBResfriamentoaaa.Append(TO_STRING(stHoraAhora.wDay));
	sSBResfriamentoaaa.Append(' ');
	sSBResfriamentoaaa.Append(TO_STRING(stHoraAhora.wHour));
	sSBResfriamentoaaa.Append(':');
	sSBResfriamentoaaa.Append(TO_STRING(stHoraAhora.wMinute));
	sSBResfriamentoaaa.Append(':');
	sSBResfriamentoaaa.Append(TO_STRING(stHoraAhora.wSecond));
	sSBResfriamentoaaa.Append('$' WHERE (`Processo` = $'');
	sSBResfriamentoaaa.Append(sGuidAtual);
	sSBResfriamentoaaa.Append('$');');
	
	sCmd := sSBResfriamentoaaa.GetString();
	
	aPara.eParaType := E_ExpParameterType.STRING_;
	aPara.nParaSize := SIZEOF(sAux);

	// call functionblock
	IF fbPLCDBRefrimaentoCmd.Execute(
		hDBID:= 1, 
		pExpression:= ADR(sCmd), 
		cbExpression:= SIZEOF(sCmd), 
		pData:= ADR(sAux), 
		cbData:= SIZEOF(sAux), 
		pParameter:= ADR(aPara), 
		cbParameter:= SIZEOF(aPara)) 
	THEN
		IF NOT fbPLCDBRefrimaentoCmd.bError THEN
			xSalvaResfriamento := FALSE;
		END_IF
	END_IF
END_IF
END_ACTION

ACTION GeraRelatorio:


fbSBaaa.Clear()
	.Append('C:\TwinCAT\n7\BaseAspercao.exe ')//C:\Users\tcuni\n7    //C:\n7\
	.Append(sGuidAtual);
	
sComando := fbSBaaa.GetString();

//Nao gera mais o relatorio aqui, agora so gera na Camara
fbProcessoEmail(
	NETID:= , 
	PATHSTR:= sComando, 
	DIRNAME:= , 
	COMNDLINE:= , 
	START:= xGeraRelatorio AND FALSE, 
	TMOUT:= , 
	BUSY=> , 
	ERR=> , 
	ERRID=> );

IF NOT fbProcessoEmail.BUSY THEN
	fbProcessoEmail.START := FALSE;
	xGeraRelatorio := FALSE;
END_IF
END_ACTION

ACTION IgnoraCarcacaBanco:


IF xSalvaIgnoraCarcaca THEN
	
	//xSalvaIgnoraCarcaca : BOOL;
	//iCarcacaIgnorada : INT;
	
	FOR i:= 0 TO 50 DO
		saAux[i]:= '';
	END_FOR
	
	//UPDATE `geral`.`carcaca` SET `Ignora` = '1' WHERE (`processo` = '{24553390-247A-46F1-9DE0-D44B8C94C4D8}' and `ncarcaca` = '1');

	saAux[0] := ('UPDATE `geral`.`carcaca` SET `Ignora` = $'1$'');
	saAux[1] := (' WHERE (`processo` = $'');
	saAux[2] := (sGuidAtual);
	saAux[3] := ('$' and `ncarcaca` = $'');
	saAux[4] := (TO_STRING(iCarcacaIgnorada));
	saAux[5] := ('$');');
	
	sCmd := F_ConcatArray(sArray:= saAux);
	
	aPara.eParaType := E_ExpParameterType.STRING_;
	aPara.nParaSize := SIZEOF(sAux);

	// call functionblock
	IF fbPLCDIgnoraCarcaca.Execute(
		hDBID:= 1, 
		pExpression:= ADR(sCmd), 
		cbExpression:= SIZEOF(sCmd), 
		pData:= ADR(sAux), 
		cbData:= SIZEOF(sAux), 
		pParameter:= ADR(aPara), 
		cbParameter:= SIZEOF(aPara)) 
	THEN
		IF NOT fbPLCDIgnoraCarcaca.bError THEN
			xSalvaIgnoraCarcaca := FALSE;
		END_IF
	END_IF
END_IF
END_ACTION

ACTION SalvaEvento:
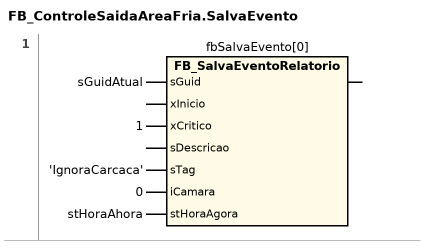
// NETWORK 1
fbSalvaEvento[0](
    sGuid := sGuidAtual,
    xCritico := 1,
    sTag := 'IgnoraCarcaca',
    iCamara := 0,
    stHoraAgora := stHoraAhora); // FB_SalvaEventoRelatorio
END_ACTION

ACTION AjustaEntrada:



iCamaraSelecionada := stFria.IHM.EN.iCamaraLiberacaoTX;
(*//DESATIVADO POR AGORA
//InternoMudou
IF stFria.c.iCamaraSelecionada <> stFriaAnterior.c.iCamaraSelecionada THEN
	iCamaraSelecionada := stFria.c.iCamaraSelecionada;
	stFria.Sup.iCamaraSelecionada := stFria.c.iCamaraSelecionada;
END_IF
//SupervisorioMudou
IF stFria.c.iCamaraSelecionada <> stFria.sup.iCamaraSelecionada THEN
	iCamaraSelecionada := stFria.Sup.iCamaraSelecionada;
	iCamaraSelecionada := stFria.Sup.iCamaraSelecionada;
END_IF
//Do Bloco mudou
IF stFria.c.iCamaraSelecionada <> iCamaraSelecionada THEN
	stFria.c.iCamaraSelecionada := iCamaraSelecionada;
	stFria.Sup.iCamaraSelecionada := iCamaraSelecionada;
END_IF
*)


IF stFria.c.xIniciaCamara <> stFriaAnterior.c.xIniciaCamara THEN
	xIniciaCamara := stFria.c.xIniciaCamara;
END_IF
IF stFria.c.xIniciaCamara <> xIniciaCamara THEN
	stFria.c.xIniciaCamara := xIniciaCamara;
END_IF

IF stFria.c.xAleatorio <> stFriaAnterior.c.xAleatorio THEN
	xAleatorio := stFria.c.xAleatorio;
END_IF
IF stFria.c.xAleatorio <> xAleatorio THEN
	stFria.c.xAleatorio := xAleatorio;
END_IF

IF stFria.c.xCapturaPeso <> stFriaAnterior.c.xCapturaPeso THEN
	xCapturaPeso := stFria.c.xCapturaPeso;
END_IF
IF stFria.c.xCapturaPeso <> xCapturaPeso THEN
	stFria.c.xCapturaPeso := xCapturaPeso;
END_IF

IF stFria.c.rPesoAtual <> stFriaAnterior.c.rPesoAtual THEN
	rPesoAtual := stFria.c.rPesoAtual;
END_IF
IF stFria.c.rPesoAtual <> rPesoAtual THEN
	stFria.c.rPesoAtual := rPesoAtual;
END_IF

IF stFria.c.xPesoNovo <> stFriaAnterior.c.xPesoNovo THEN
	xPesoNovo := stFria.c.xPesoNovo;
END_IF
IF stFria.c.xPesoNovo <> xPesoNovo THEN
	stFria.c.xPesoNovo := xPesoNovo;
END_IF





stFriaAnterior := stFria;
END_ACTION

ACTION AjustaSaida:




stFria.c.iCamarasDisponiveis := iCamarasDisponiveis;
//stIHM.rPesosQuentes := rPesosQuentes;
//stIHM.rPesosfrios := rPesosFrios;
stFria.c.sGuidAtual := sGuidAtual;
stFria.c.iCarcacaAtual := iCarcacaAtual;


stFria.ihm.SA.xCamaraSelecionadaLiberadaRX := xCamaraSelecionadaOK;
stFria.IHM.SA.rPesoFrioAtualRX := rPesoAtual;
stFria.ihm.SA.xEmProcesso := stFria.C.xEmProcesso;
stFria.ihm.SA.iAmostraAtualRX := iCarcacaAtual;
stFria.ihm.SA.iQtdAmostradaRX := iCarcacaAtual-1;
stFria.ihm.SA.iFaltaAmostrarRX := iNumeroAmostras - (iCarcacaAtual-1);

stFria.Sup.iCarcacasAmostradas := iCarcacaAtual-1;
stFria.Sup.iCarcacasFaltaAmostrar := iNumeroAmostras - (iCarcacaAtual-1);
stFria.Sup.iCarcacasAmostragemTotal := iNumeroAmostras;


FOR i := 0 TO 50 DO
	//Esse if so existe pq ta dando exception quando entra online aqui, nao faz o menor sentido
	IF  iCamarasDisponiveis[i] > 0 AND iCamarasDisponiveis[i] < 100 THEN
		stFria.Sup.stCamarasDisponiveis[i].iCamara := iCamarasDisponiveis[i];
		stFria.Sup.stCamarasDisponiveis[i].sNome := stCamaras[iCamarasDisponiveis[i]].config.sNome;
	END_IF
END_FOR


FOR i := 1 TO 20 DO
	IF xCacacasIgnoradas[i] THEN
		stFria.IHM.SA.sPesoCaraca[i] := 'Ignorada';
		stFria.IHM.SA.iCarcacaIgnorada[i] := 2;
	ELSE
		stFria.IHM.SA.sPesoCaraca[i] := TO_STRING(rPesosFrios[i]);
		IF rPesosFrios[i] > 5 THEN
			stFria.IHM.SA.iCarcacaIgnorada[i] := 1;
		ELSE
			stFria.IHM.SA.iCarcacaIgnorada[i] := 0;
		END_IF
	END_IF
	
END_FOR
END_ACTION

ACTION PegaCamarasDisponiveis:




iMinCamaras := (LOWER_BOUND(stCamaras,1));
iMaxCamaras := (UPPER_BOUND(stCamaras,1));

IF iMinCamaras > iMaxCamaras THEN
	diaux := iMinCamaras;
	iMinCamaras := iMaxCamaras;
	iMaxCamaras := diaux;
END_IF

FOR i := 0 TO 50 DO
	iCamarasDisponiveis[i] := 0;
END_FOR

iAux := 0;
FOR i := DINT_TO_INT(iMinCamaras) TO DINT_TO_INT(iMaxCamaras) DO
	IF stCamaras[i].en.sGuidAtual <> '' AND stCamaras[i].status.xTerminouAspercao THEN
		iCamarasDisponiveis[iAux] := stCamaras[i].config.iCamara;
		iAux := iAux + 1;
	END_IF
END_FOR

j;
END_ACTION

ACTION VeCarcacasAIgnorar:




FOR i := 1 TO 20 DO
	rtCacacasAIgnorar[i](CLK:= stFria.IHM.EN.xIgnoraCarcaca[i], Q=> );	
	IF rtCacacasAIgnorar[i].Q THEN
		xCacacasIgnoradas[i] := TRUE;
		//Salva no banco
		xSalvaIgnoraCarcaca := TRUE;
		iCarcacaIgnorada := i;
		//Garante que vai ficar zerado esse cara
		rPesosFrios[i] := 0;
		rPesosQuentes[i] := 0;
	END_IF
END_FOR
END_ACTION

END_FUNCTION_BLOCK

// POUs/Automatico/Aspercao/ControleLiberacaoCamaras/AreaQuente/FB_ControleEntradaAreaQuente
FUNCTION_BLOCK FB_ControleEntradaAreaQuente
VAR_IN_OUT
	stAreaQuente : st_areaquente;
	stCamaras : ARRAY[*] OF st_Camara;
END_VAR
VAR_INPUT
	iCamaraSelecionada	: INT;// qual camara o operador escolher para começar
	xIniciaCamara		: BOOL;// operador dizendo para começar a amostragem
	xAleatorio			: BOOL;// se vai fazer a amostragem aleatorio ou sequencial
	xCapturaPeso		: BOOL;// operador dizendo para pegar o peso atual
	rPesoAtual			: REAL;// Peso atual que vem da balança
	xPesoNovo			: BOOL;// Quando  balança diz que veio um peso novo
	stHoraAhora 		: TIMESTRUCT; //Hora atual 
END_VAR
VAR_OUTPUT
	iCamarasDisponiveis : ARRAY[0..50] OF INT; // para a lista do cara para escolher a camara
	rPesosQuentes		: ARRAY[0..1000] OF REAL; // 	array com os pesos quentes amostrados pelo operador ou sequencialmente
	sGuidAtual			: STRING;// guid do processo atual
	iCarcacaAtual		: INT;// Qual o numero da carcaça que ele ta esperando
	xCamaraSelecionadaOK : BOOL;//se a camara selecionada pode entrar porco
	xEmProcesso			: BOOL;
	xPesoColetadoRX		: BOOL;
	iNumeroAmostras 	: INT;
END_VAR
VAR
	sSBaasdaeuteodeio2		  : FB_StringBuilder;
	
	
	stAnterior  : st_areaquente;
	fbCriaGUID 	: FB_CreateGUID;
	xCriaGuid 	: BOOL;
	guidCriado 	: Guid;
	
	iMinCamaras : DINT;
	iMaxCamaras : DINT;
	
	i : INT;
	iAux : INT;
	
	iEstado : INT;
	
	
	//grava o novo processo
	fbPLCDBWrite		: FB_PLCDBWriteEvt(sNetID := '', tTimeout := T#3S); //Bloco para gravar no banco de dados
	xGravaProcesso		: BOOL;
	EstruturaBanco 		: st_ProcessoBD;
	ColumnNamesGrava 	: ARRAY[0..14] OF STRING(50) := ['Processo',
														'Camara',
														'InicioResfriamento',
														'FimResfriamento',
														'InicioAspersao',
														'FimAspersao',
														'NumeroCarcacas',
														'ConsumoAguaTotal',
														'Cancelado',
														'Finalizado',
														'Aspergida',
														'Pesoquente',
														'PesoFrio',
														'Status',
														'Timestamp'];
														
	//grava nova carcaca
	xGravaCarcaca			: BOOL;
	xGravaPesoQuente		: BOOL;
	EstruturaBancoCarcaca 	: st_CarcacaBD;
						
    fbPLCDBCmd    : FB_PLCDBCmdEvt(sNetID := '', tTimeout := T#2S);
    sCmd          : STRING (1000); 
    aPara         : ST_ExpParameter;
	sAux 		  : STRING;
	
	stTSAux 	  : TIMESTRUCT; //Hora atual 
	
	rPesoQuentetotal : REAL;
	
	diaux : DINT;
	
	rtNovoPeso : r_TRIG;
	btNovoPeso : b_TRIG;
	rtNovaCaptura : r_TRIG;
	
	
	xAmostraProximoPeso : BOOL;
	xSalvaAmostra : BOOL;
	
	rtCancela : R_TRIG;
	xCancela : BOOL;
	xTeste : BOOL;
	
END_VAR

IF TRUE THEN

	AjustaEntrada();
	PegaCamarasDisponiveis();
	
	//Se o cara quiser cancelar a aquisição
	rtCancela(CLK:= stAreaQuente.c.xCancela, Q=> );
	IF rtCancela.q THEN
		xCancela := TRUE;
	END_IF
	Cancela();
	
	CASE iEstado OF
		0://Esperando
		//fazer esquema pra ver se a camara selecionada esta dentro das que da pra selecionar
		
			xCamaraSelecionadaOK := FALSE;
			FOR i := 0 TO 50 DO
				IF iCamarasDisponiveis[i]  = 0 THEN
					EXIT;
				ELSE
					xCamaraSelecionadaOK := xCamaraSelecionadaOK OR iCamaraSelecionada = iCamarasDisponiveis[i];
				END_IF
			END_FOR
			
			
			IF xCamaraSelecionadaOK AND (xIniciaCamara OR stAreaQuente.Sup.xIniciarAmostragem OR stAreaQuente.ihm.EN.xIniciaCamaraTX OR stAreaQuente.ihm.EN.xIniciaAmostragemSequencialTX) THEN
				iEstado := 1;
				xIniciaCamara := FALSE;
				xEmProcesso := TRUE;
				stAreaQuente.Sup.xIniciarAmostragem := FALSE;
			END_IF
		
		1://Cria guid e vai para amostrar as carcaças
			xCriaGuid := TRUE;
			fbCriaGUID(
				bExecute:= xCriaGuid, 
				sNetId:= '', 
				tTimeout:= T#5S, 
				pGuidBuffer:= ADR(guidCriado), 
				nGuidBufferSize:= SIZEOF(guidCriado), 
				bBusy=> , 
				bError=> , 
				nErrorId=> );
			
			IF NOT fbCriaGUID.bBusy THEN
				xCriaGuid := FALSE;
				sGuidAtual := GUID_TO_REGSTRING(guidCriado);
				stCamaras[iCamaraSelecionada].en.sGuidAtual := sGuidAtual;
				stCamaras[iCamaraSelecionada].Status.xPegandoPesosQuentes := TRUE;
				iNumeroAmostras := stCamaras[iCamaraSelecionada].config.iCarcacasReal;
				iEstado := 2;
				xGravaProcesso := TRUE;
				fbCriaGUID(bExecute:= FALSE);
			END_IF
		
		2://Cria o processo
		
			EstruturaBanco.Processo 	:= sGuidAtual;
			EstruturaBanco.Camara 		:= iCamaraSelecionada;
			EstruturaBanco.Status 		:= 'Aquisitando carcaças';
			EstruturaBanco.Timestamp 	:= SYSTEMTIME_TO_DT(stHoraAhora);
			
			EscreveNovoProcessoBanco();
			
			IF NOT xGravaProcesso THEN
				
				iNumeroAmostras := stCamaras[iCamaraSelecionada].config.iCarcacasAmostra;
				iCarcacaAtual := 1;
				
				
				CASE stAreaQuente.Sup.iModoDeAmostragem OF
					1://RFID
					2://Consecutivo
						iEstado := 3;
					3://Manual/Aleatorio
						iEstado := 6;
					4://ForaDoSistema, quando ta fora ele amostra 0 carcaças e ja eras
						iEstado := 3;
						iNumeroAmostras := 0;
				END_CASE
				
				btNovoPeso(CLK:= xPesoNovo, Q=> );
				rtNovaCaptura(CLK:= xCapturaPeso OR stAreaQuente.Sup.xCapturaAmostra OR stAreaQuente.ihm.EN.xColetaAmostraTX, Q=> );
			END_IF
			
			
		3://Peso sequencial
			//quando der as 20 camaras e nao tiver carregando a camara ele nao vai pro fim
			IF iCarcacaAtual > iNumeroAmostras AND NOT xIniciaCamara THEN
				iEstado := 5;
				xGravaPesoQuente := TRUE;
			END_IF
			
			rtNovoPeso(CLK:= xPesoNovo OR xTeste OR stAreaQuente.Sup.xNovoPesoDebug, Q=> );
			
			//Ajusta o peso caso ele seja por debug
			IF rtNovoPeso.q THEN
				IF stAreaQuente.Sup.xNovoPesoDebug THEN
					rPesoAtual := stAreaQuente.Sup.rPesoDebug;
				END_IF
			END_IF
			
			
			IF  rtNovoPeso.q AND
				rPesoAtual > 3 AND // so garante que o peso nao é zero nem muito baixo
				iCarcacaAtual < iNumeroAmostras + 1 // garante que nao vai ficar adicionando carcaça alem do que precisa
				THEN 
			   
				rPesosQuentes[iCarcacaAtual] := rPesoAtual;
				iEstado := 4;
				xGravaCarcaca := TRUE;
			END_IF
			
			
		6://Peso manual
			//quando der as 20 camaras e nao tiver carregando a camara ele nao vai pro fim
			IF iCarcacaAtual > iNumeroAmostras AND NOT xIniciaCamara THEN
				iEstado := 5;
				xGravaPesoQuente := TRUE;
			END_IF
			
			rtNovaCaptura(CLK:= xCapturaPeso OR stAreaQuente.Sup.xCapturaAmostra OR stAreaQuente.ihm.EN.xColetaAmostraTX, Q=> );
			IF rtNovaCaptura.q THEN
				xAmostraProximoPeso := TRUE;
			END_IF
			
			rtNovoPeso(CLK:= xPesoNovo OR stAreaQuente.Sup.xNovoPesoDebug, Q=> );
			IF rtNovoPeso.q AND xAmostraProximoPeso THEN
				xSalvaAmostra := TRUE;
			END_IF
			
			
			IF xSalvaAmostra  AND
				rPesoAtual > 3 AND // so garante que o peso nao é zero nem muito baixo
				iCarcacaAtual < iNumeroAmostras+ 1 // garante que nao vai ficar adicionando carcaça alem do que precisa
				THEN 
			   
				xPesoColetadoRX := TRUE;
				xSalvaAmostra := FALSE;
				xAmostraProximoPeso := FALSE;
				rPesosQuentes[iCarcacaAtual] := rPesoAtual;
				iEstado := 4;
				xGravaCarcaca := TRUE;
			END_IF
			
			
		4: //Salva no banco essa carcaça
		
			EstruturaBancoCarcaca.Camara 		:= iCamaraSelecionada;
			EstruturaBancoCarcaca.Processo 		:= sGuidAtual;
			EstruturaBancoCarcaca.nCarcaca 		:= iCarcacaAtual;
			EstruturaBancoCarcaca.PesoQuente	:= rPesosQuentes[iCarcacaAtual];
			
			EstruturaBancoCarcaca.Status 		:= 'Esperando asperção';
			
			EscreveNovaCarcacaBanco();
			
			
			IF NOT xGravaCarcaca THEN
				xPesoColetadoRX := FALSE;
				IF xAleatorio THEN
					iEstado := 6;
				ELSE
					iEstado := 3;
				END_IF
				
				iCarcacaAtual := iCarcacaAtual + 1;
			END_IF
		
		
		5://Soma os pesos quentes e salva no processo
			EscrevePesoQuenteProcesso();
			
			IF NOT xGravaPesoQuente THEN
				
				stCamaras[iCamaraSelecionada].en.rPesosQuente := rPesosQuentes;
				stCamaras[iCamaraSelecionada].Status.xPegandoPesosQuentes := FALSE;
			
				//Volta pro inicio e deixa tudo pronto para o proximo ciclo
				iEstado := 0;
				FOR i := 1 TO iNumeroAmostras DO
					rPesosQuentes[i] := 0;
				END_FOR
				sGuidAtual := '';
				iCamaraSelecionada := 0;
				iCarcacaAtual := 1;
				xEmProcesso := FALSE;
			END_IF
		
		
	END_CASE
	
	
	
	
	
	
	
	AjustaSaida();
	

END_IF

ACTION Cancela:



//UPDATE `geral`.`processos` SET `Cancelado` = '1' WHERE (`Processo` = 'teste');



IF xCancela THEN
	sSBaasdaeuteodeio2.Clear();
	sSBaasdaeuteodeio2.Append('UPDATE `geral`.`processos` SET `Cancelado` = $'1$' WHERE (`Processo` = $'');
	sSBaasdaeuteodeio2.Append(sGuidAtual);
	sSBaasdaeuteodeio2.Append(')$';');
	
	sCmd := sSBaasdaeuteodeio2.GetString();
	
	aPara.eParaType := E_ExpParameterType.STRING_;
	aPara.nParaSize := SIZEOF(sAux);

	// call functionblock
	IF fbPLCDBCmd.Execute(
		hDBID:= 1, 
		pExpression:= ADR(sCmd), 
		cbExpression:= SIZEOF(sCmd), 
		pData:= ADR(sAux), 
		cbData:= SIZEOF(sAux), 
		pParameter:= ADR(aPara), 
		cbParameter:= SIZEOF(aPara)) 
	THEN
		xCancela := FALSE;
		sGuidAtual := '';
		stCamaras[iCamaraSelecionada].en.sGuidAtual := sGuidAtual;
		iEstado := 0;
		
		FOR i := 1 TO 20 DO
			rPesosQuentes[i] := 0;
		END_FOR
		
		iCamaraSelecionada := 0;
		xEmProcesso := FALSE;
	END_IF
END_IF
END_ACTION

ACTION EscreveNovaCarcacaBanco:

		
IF xGravaCarcaca THEN
	sSBaasdaeuteodeio2.Clear();
	sSBaasdaeuteodeio2.Append('INSERT INTO `geral`.`carcaca` (`Camara`, `Processo`, `nCarcaca`, `PesoQuente`, `horaPesoQuente`, `Status`) VALUES ($'');
	sSBaasdaeuteodeio2.Append(TO_STRING(EstruturaBancoCarcaca.Camara));
	sSBaasdaeuteodeio2.Append('$', $'');
	sSBaasdaeuteodeio2.Append(TO_STRING(EstruturaBancoCarcaca.Processo));
	sSBaasdaeuteodeio2.Append('$', $'');
	sSBaasdaeuteodeio2.Append(TO_STRING(EstruturaBancoCarcaca.nCarcaca));
	sSBaasdaeuteodeio2.Append('$', $'');
	sSBaasdaeuteodeio2.Append(TO_STRING(EstruturaBancoCarcaca.PesoQuente));
	sSBaasdaeuteodeio2.Append('$', $'');
	sSBaasdaeuteodeio2.Append(TO_STRING(stHoraAhora.wYear));
	sSBaasdaeuteodeio2.Append('-');
	sSBaasdaeuteodeio2.Append(TO_STRING(stHoraAhora.wMonth));
	sSBaasdaeuteodeio2.Append('-');
	sSBaasdaeuteodeio2.Append(TO_STRING(stHoraAhora.wDay));
	sSBaasdaeuteodeio2.Append(' ');
	sSBaasdaeuteodeio2.Append(TO_STRING(stHoraAhora.wHour));
	sSBaasdaeuteodeio2.Append(':');
	sSBaasdaeuteodeio2.Append(TO_STRING(stHoraAhora.wMinute));
	sSBaasdaeuteodeio2.Append(':');
	sSBaasdaeuteodeio2.Append(TO_STRING(stHoraAhora.wSecond));
	sSBaasdaeuteodeio2.Append('$', $'');
	sSBaasdaeuteodeio2.Append(TO_STRING(EstruturaBancoCarcaca.Status));
	sSBaasdaeuteodeio2.Append('$');');
	
	sCmd := sSBaasdaeuteodeio2.GetString();
	
	aPara.eParaType := E_ExpParameterType.STRING_;
	aPara.nParaSize := SIZEOF(sAux);

	// call functionblock
	IF fbPLCDBCmd.Execute(
		hDBID:= 1, 
		pExpression:= ADR(sCmd), 
		cbExpression:= SIZEOF(sCmd), 
		pData:= ADR(sAux), 
		cbData:= SIZEOF(sAux), 
		pParameter:= ADR(aPara), 
		cbParameter:= SIZEOF(aPara)) 
	THEN	
		IF NOT fbPLCDBCmd.bError THEN
			xGravaCarcaca := FALSE;
		END_IF
	END_IF
END_IF
END_ACTION

ACTION EscreveNovoProcessoBanco:


///INSERT INTO `geral`.`processos` (`Processo`, `Camara`, `Status`, `Timestamp`) VALUES ('sd', 'dd', 'dd', 'asd');

IF xGravaProcesso THEN
	
	sSBaasdaeuteodeio2.Clear();
	sSBaasdaeuteodeio2.Append('INSERT INTO `geral`.`processos` (`Processo`, `Camara`, `Status`, `Timestamp`) VALUES ($'');
	sSBaasdaeuteodeio2.Append(TO_STRING(EstruturaBanco.Processo));
	sSBaasdaeuteodeio2.Append('$', $'');
	sSBaasdaeuteodeio2.Append(TO_STRING(EstruturaBanco.Camara));
	sSBaasdaeuteodeio2.Append('$', $'');
	sSBaasdaeuteodeio2.Append(TO_STRING(EstruturaBanco.Status));
	sSBaasdaeuteodeio2.Append('$', $'');
	sSBaasdaeuteodeio2.Append(TO_STRING(stHoraAhora.wYear));
	sSBaasdaeuteodeio2.Append('-');
	sSBaasdaeuteodeio2.Append(TO_STRING(stHoraAhora.wMonth));
	sSBaasdaeuteodeio2.Append('-');
	sSBaasdaeuteodeio2.Append(TO_STRING(stHoraAhora.wDay));
	sSBaasdaeuteodeio2.Append(' ');
	sSBaasdaeuteodeio2.Append(TO_STRING(stHoraAhora.wHour));
	sSBaasdaeuteodeio2.Append(':');
	sSBaasdaeuteodeio2.Append(TO_STRING(stHoraAhora.wMinute));
	sSBaasdaeuteodeio2.Append(':');
	sSBaasdaeuteodeio2.Append(TO_STRING(stHoraAhora.wSecond));
	sSBaasdaeuteodeio2.Append('$');');
	
	sCmd := sSBaasdaeuteodeio2.GetString();
	
	aPara.eParaType := E_ExpParameterType.STRING_;
	aPara.nParaSize := SIZEOF(sAux);

	// call functionblock
	IF fbPLCDBCmd.Execute(
		hDBID:= 1, 
		pExpression:= ADR(sCmd), 
		cbExpression:= SIZEOF(sCmd), 
		pData:= ADR(sAux), 
		cbData:= SIZEOF(sAux), 
		pParameter:= ADR(aPara), 
		cbParameter:= SIZEOF(aPara)) 
	THEN
		IF NOT fbPLCDBCmd.bError THEN
			xGravaProcesso := FALSE;
		END_IF
	END_IF
END_IF
END_ACTION

ACTION EscrevePesoQuenteProcesso:


		
IF xGravaPesoQuente THEN
	rPesoQuentetotal := 0;
	
	FOR i := 1 TO 20 DO
		rPesoQuentetotal := rPesoQuentetotal + rPesosQuentes[i];
	END_FOR



	sSBaasdaeuteodeio2.Clear();
	sSBaasdaeuteodeio2.Append('UPDATE `geral`.`processos` SET `Pesoquente` = $'');
	sSBaasdaeuteodeio2.Append(TO_STRING(rPesoQuentetotal));
	sSBaasdaeuteodeio2.Append('$', `Status` = $'Peso quente concluido / Esperando asperção');
	sSBaasdaeuteodeio2.Append('$' WHERE (`Processo` = $'');
	sSBaasdaeuteodeio2.Append(sGuidAtual);
	sSBaasdaeuteodeio2.Append('$');');
	
	sCmd := sSBaasdaeuteodeio2.GetString();
	
	aPara.eParaType := E_ExpParameterType.STRING_;
	aPara.nParaSize := SIZEOF(sAux);

	// call functionblock
	IF fbPLCDBCmd.Execute(
		hDBID:= 1, 
		pExpression:= ADR(sCmd), 
		cbExpression:= SIZEOF(sCmd), 
		pData:= ADR(sAux), 
		cbData:= SIZEOF(sAux), 
		pParameter:= ADR(aPara), 
		cbParameter:= SIZEOF(aPara)) 
	THEN	
		IF NOT fbPLCDBCmd.bError THEN
			xGravaPesoQuente := FALSE;
		END_IF
	END_IF
END_IF
END_ACTION

ACTION AjustaEntrada:




iCamaraSelecionada := stAreaQuente.IHM.EN.iCamaraCarregementoTX;
(*//DESATIVADO POR AGORA
//InternoMudou
IF stAreaQuente.c.iCamaraSelecionada <> stAnterior.c.iCamaraSelecionada THEN
	iCamaraSelecionada := stAreaQuente.c.iCamaraSelecionada;
	stAreaQuente.Sup.iCamaraSelecionada := stAreaQuente.c.iCamaraSelecionada;
END_IF
//SupervisorioMudou/
IF stAreaQuente.c.iCamaraSelecionada <> stAreaQuente.Sup.iCamaraSelecionada AND FALSE THEN
	iCamaraSelecionada := stAreaQuente.Sup.iCamaraSelecionada;
	iCamaraSelecionada := stAreaQuente.Sup.iCamaraSelecionada;
END_IF
//Do Bloco mudou
IF stAreaQuente.c.iCamaraSelecionada <> iCamaraSelecionada THEN
	stAreaQuente.c.iCamaraSelecionada := iCamaraSelecionada;
	stAreaQuente.Sup.iCamaraSelecionada := iCamaraSelecionada;
END_IF
*)






IF stAreaQuente.c.xIniciaCamara <> stAnterior.c.xIniciaCamara THEN
	xIniciaCamara := stAreaQuente.c.xIniciaCamara;
END_IF
IF stAreaQuente.c.xIniciaCamara <> xIniciaCamara THEN
	stAreaQuente.c.xIniciaCamara := xIniciaCamara;
END_IF

IF stAreaQuente.c.xAleatorio <> stAnterior.c.xAleatorio THEN
	xAleatorio := stAreaQuente.c.xAleatorio;
END_IF
IF stAreaQuente.c.xAleatorio <> xAleatorio THEN
	stAreaQuente.c.xAleatorio := xAleatorio;
END_IF

IF stAreaQuente.c.xCapturaPeso <> stAnterior.c.xCapturaPeso THEN
	xCapturaPeso := stAreaQuente.c.xCapturaPeso;
END_IF
IF stAreaQuente.c.xCapturaPeso <> xCapturaPeso THEN
	stAreaQuente.c.xCapturaPeso := xCapturaPeso;
END_IF

IF stAreaQuente.c.rPesoAtual <> stAnterior.c.rPesoAtual THEN
	rPesoAtual := stAreaQuente.c.rPesoAtual;
END_IF
IF stAreaQuente.c.rPesoAtual <> rPesoAtual THEN
	stAreaQuente.c.rPesoAtual := rPesoAtual;
END_IF

IF stAreaQuente.c.xPesoNovo <> stAnterior.c.xPesoNovo THEN
	xPesoNovo := stAreaQuente.c.xPesoNovo;
END_IF
IF stAreaQuente.c.xPesoNovo <> xPesoNovo THEN
	stAreaQuente.c.xPesoNovo := xPesoNovo;
END_IF





stAnterior := stAreaQuente;
END_ACTION

ACTION AjustaSaida:




stAreaQuente.c.iCamarasDisponiveis := iCamarasDisponiveis;
//stIHM.rPesosQuentes := rPesosQuentes;
stAreaQuente.c.sGuidAtual := sGuidAtual;
stAreaQuente.c.iCarcacaAtual := iCarcacaAtual;
stAreaQuente.c.xEmProcesso := xEmProcesso;
stAreaQuente.c.xPesoColetadoRX := xPesoColetadoRX;


stAreaQuente.ihm.SA.xCamaraSelecionadaLiberadaRX := xCamaraSelecionadaOK;
stAreaQuente.IHM.SA.rPesoQuenteAtualRX := rPesoAtual;
stAreaQuente.ihm.SA.xEmProcesso := xEmProcesso;
stAreaQuente.ihm.SA.iAmostraAtualRX := iCarcacaAtual;
stAreaQuente.ihm.SA.iQtdAmostradaRX := iCarcacaAtual-1;
stAreaQuente.ihm.SA.iFaltaAmostrarRX := iNumeroAmostras - (iCarcacaAtual-1);


stAreaQuente.Sup.iCarcacasAmostradas := iCarcacaAtual-1;
stAreaQuente.Sup.iCarcacasFaltaAmostrar := iNumeroAmostras - (iCarcacaAtual-1);
stAreaQuente.Sup.iCarcacasAmostragemTotal := iNumeroAmostras;


FOR i := 0 TO 50 DO
	//Esse if so existe pq ta dando exception quando entra online aqui, nao faz o menor sentido
	IF  iCamarasDisponiveis[i] > 0 AND iCamarasDisponiveis[i] < 100 THEN
		stAreaQuente.Sup.stCamarasDisponiveis[i].iCamara := iCamarasDisponiveis[i];
		stAreaQuente.Sup.stCamarasDisponiveis[i].sNome := stCamaras[iCamarasDisponiveis[i]].config.sNome;
	END_IF
END_FOR
END_ACTION

ACTION PegaCamarasDisponiveis:




//iMinCamaras := (LOWER_BOUND(stCamaras,1));
//iMaxCamaras := (UPPER_BOUND(stCamaras,1));

iMinCamaras := 0;
iMaxCamaras := 60;

IF iMinCamaras > iMaxCamaras THEN
	diaux := iMinCamaras;
	iMinCamaras := iMaxCamaras;
	iMaxCamaras := diaux;
END_IF


FOR i := 0 TO 50 DO
	iCamarasDisponiveis[i] := 0;
END_FOR

iAux := 0;
FOR i := DINT_TO_INT(iMinCamaras) TO DINT_TO_INT(iMaxCamaras) DO
	IF stCamaras[i].en.sGuidAtual = '' AND stCamaras[i].config.sValvulas <> '' THEN
		iCamarasDisponiveis[iAux] := stCamaras[i].config.iCamara;
		iAux := iAux + 1;
	END_IF
END_FOR
END_ACTION

END_FUNCTION_BLOCK

// POUs/Automatico/Aspercao/ControleProtocolo/FB_ControleEdicaoProtocolo
FUNCTION_BLOCK FB_ControleEdicaoProtocolo
VAR_IN_OUT
	Protocolos : ARRAY[*] OF st_Protocolo;//de 0 a um valor x menor que 1000
	sNomeProtocoloIHM : ARRAY[*] OF STRING;//de 0 a um valor x menor que 1000
	stControle : ARRAY[*] OF st_ControleValvula;//de 0 a um valor x menor que 1000
	stCamara : ARRAY[*] OF st_Camara;//de 0 a um valor x menor que 1000
END_VAR
VAR_INPUT
	xLeDoBanco : BOOL;
	sNomeTabela : STRING := 'protocolo';
	xProtocoloPorCamara : BOOL;
END_VAR
VAR_OUTPUT
	xOcupado : BOOL;
	iEstado : INT;
END_VAR
VAR
	uiBaixoArray : DINT;
	uiCimaArray : DINT;
	
	uiBaixoArraystControle : DINT;
	uiCimaArraystControle : DINT;
	
	stEstruturasBanco : ARRAY[0..1000] OF st_DBProtocolo;
	
	fbPLCDBRead		: FB_PLCDBReadEvt(sNetID := '', tTimeout := T#3M); //Bloco para leitura do banco de dados sem filtro
	ColumnNamesLe 	: ARRAY[0..34] OF STRING(50) := ['ID',
													'Nome',
													'NomeIHM',
													'Valvulas',
													'ET01TON',
													'ET01TOFF',
													'ET01NC',
													'ET02TON',
													'ET02TOFF',
													'ET02NC',
													'ET03TON',
													'ET03TOFF',
													'ET03NC',
													'ET04TON',
													'ET04TOFF',
													'ET04NC',
													'ET05TON',
													'ET05TOFF',
													'ET05NC',
													'ET06TON',
													'ET06TOFF',
													'ET06NC',
													'ET07TON',
													'ET07TOFF',
													'ET07NC',
													'ET08TON',
													'ET08TOFF',
													'ET08NC',
													'ET09TON',
													'ET09TOFF',
													'ET09NC',
													'ET10TON',
													'ET10TOFF',
													'ET10NC',
													'xFinalDeSemana'];
													
													
	sCmdUpdate : STRING(5000);
	fbPLCDBCmd    : FB_PLCDBCmdEvt(sNetID := '', tTimeout := T#5S);
	aPara : ST_ExpParameter;
	
	
	
	fbDataBase 	:	FB_SQLDatabaseEvt('',T#5S);
	fbComando	:	FB_SQLCommandEvt('',T#5S);
	fbResultado	:	FB_SQLResultEvt('',T#5S);
	sCmd		: 	STRING(1000);
	
	i : INT;
	j : INT;
	k : INT;
	iProtocoloAlterado : INT;
	
	fbSB		: FB_StringBuilder;
	sAux 		: ARRAY[0..15] OF STRING(80);
	
	sAuxVazio 	: STRING;
	
	iValvulas 	: ARRAY[0..500] OF INT;
	
	ProtocoloVazio : st_Protocolo;
	
END_VAR




IF xLicensaValida6446896834 THEN	

	uiCimaArray		:= UPPER_BOUND(Protocolos, 1);
	uiBaixoArray	:= LOWER_BOUND(Protocolos, 1);
	
	CASE iEstado OF 
	
		0 : //começa sem os valores e passa no banco pra ver como ta
		
		IF xLeDoBanco THEN
			xOcupado := TRUE;
			IF fbPLCDBRead.ReadStruct(
										hDBID:=1 , 
										sTableName:= sNomeTabela, 
										pColumnNames:= ADR(ColumnNamesLe), 
										cbColumnNames:= SIZEOF(ColumnNamesLe), 
										sOrderByColumn:= ColumnNamesLe[0], 
										eOrderType:= E_OrderType.ASC, 
										nStartIndex:= uiBaixoArray, 
										nRecordCount:= uiCimaArray-uiBaixoArray+1, 
										pData:= ADR(stEstruturasBanco), 
										cbData:= SIZEOF(stEstruturasBanco))
				THEN
					iEstado := 1;	
					xLeDoBanco := FALSE;
				END_IF
					
			uiCimaArraystControle	:= UPPER_BOUND(stControle, 1);
			uiBaixoArraystControle	:= LOWER_BOUND(stControle, 1);
			FOR i := DINT_TO_INT(uiBaixoArray) TO DINT_TO_INT(uiCimaArray) DO
				Protocolos[i].DB := stEstruturasBanco[i];
			END_FOR
			
		END_IF
			
		1:// vai trabalhar os dados que vieram de quando leu o banco e vai atualizar o que tem no array da estrutura
		
		IF NOT xProtocoloPorCamara THEN
			
			uiCimaArraystControle	:= UPPER_BOUND(stControle, 1);
			uiBaixoArraystControle	:= LOWER_BOUND(stControle, 1);
			FOR i := DINT_TO_INT(uiBaixoArraystControle) TO DINT_TO_INT(uiCimaArraystControle) DO
				stControle[i].EN.sIHM[0] := '';
				stControle[i].EN.sIHM[1] := '';
				stControle[i].EN.sIHM[2] := '';
				stControle[i].EN.sIHM[3] := '';
			END_FOR
			
			
			FOR i := DINT_TO_INT(uiBaixoArray) TO DINT_TO_INT(uiCimaArray) DO
				//Protocolos[i].DB := stEstruturasBanco[i];
				sNomeProtocoloIHM[i] := CONCAT(DINT_TO_STRING(Protocolos[i].DB.ID),CONCAT(' - ',Protocolos[i].DB.Nome));
				//do protocolo rodando ve quais as valvulas nele
				F_StringSeparadorFBGrupos(sStr:= Protocolos[i].DB.Valvulas, ListaINT:=iValvulas);
				//roda todas as valvulas no protocolo
				FOR j := 0 TO 500 DO
					IF iValvulas[j] = 0 THEN
						EXIT;
					END_IF
					//encontra uma posição vazia no role
					FOR k := 0 TO 3 DO
						IF stControle[iValvulas[j]].EN.sIHM[k] = '' THEN
							EXIT;
						END_IF
					END_FOR
					//se for > 3 siginifica que ja ocupou todas as posiçoes
					IF k < 3 THEN
						//joga o protocolo na posiçao vazia e o nome na posiçao vazia
						CASE k OF
							0:
								stControle[iValvulas[j]].EN.stProtocolos[0] := Protocolos[i];
								stControle[iValvulas[j]].EN.sIHM[0] := Protocolos[i].DB.NomeIHM;
							1:
								stControle[iValvulas[j]].EN.stProtocolos[1] := Protocolos[i];
								stControle[iValvulas[j]].EN.sIHM[1] := Protocolos[i].DB.NomeIHM;
							2:
								stControle[iValvulas[j]].EN.stProtocolos[2] := Protocolos[i];
								stControle[iValvulas[j]].EN.sIHM[2] := Protocolos[i].DB.NomeIHM;
							3:
								stControle[iValvulas[j]].EN.stProtocolos[3] := Protocolos[i];
								stControle[iValvulas[j]].EN.sIHM[3] := Protocolos[i].DB.NomeIHM;
						END_CASE
					END_IF
				END_FOR
			END_FOR
		ELSE
			//aqui manda o protocolo para a camara
			uiCimaArraystControle	:= UPPER_BOUND(stCamara, 1);
			uiBaixoArraystControle	:= LOWER_BOUND(stCamara, 1);
			//limpa os protocolos das camaras
			FOR i := TO_INT(uiBaixoArraystControle) TO TO_INT(uiCimaArraystControle) DO
				FOR j := 0 TO 30 DO
					stCamara[i].config.stProtocolos[j] := ProtocoloVazio;
				END_FOR
			END_FOR
			
			FOR i := DINT_TO_INT(uiBaixoArraystControle) TO DINT_TO_INT(uiCimaArraystControle) DO
				FOR j := 0 TO 30 DO
					CASE j OF
						0:stCamara[i].config.stProtocolos[0] := Protocolos[j];
						1:stCamara[i].config.stProtocolos[1] := Protocolos[j];
						2:stCamara[i].config.stProtocolos[2] := Protocolos[j];
						3:stCamara[i].config.stProtocolos[3] := Protocolos[j];
						4:stCamara[i].config.stProtocolos[4] := Protocolos[j];
						5:stCamara[i].config.stProtocolos[5] := Protocolos[j];
						6:stCamara[i].config.stProtocolos[6] := Protocolos[j];
						7:stCamara[i].config.stProtocolos[7] := Protocolos[j];
						8:stCamara[i].config.stProtocolos[8] := Protocolos[j];
						9:stCamara[i].config.stProtocolos[9] := Protocolos[j];
						10:stCamara[i].config.stProtocolos[10] := Protocolos[j];
						11:stCamara[i].config.stProtocolos[11] := Protocolos[j];
						12:stCamara[i].config.stProtocolos[12] := Protocolos[j];
						13:stCamara[i].config.stProtocolos[13] := Protocolos[j];
						14:stCamara[i].config.stProtocolos[14] := Protocolos[j];
						15:stCamara[i].config.stProtocolos[15] := Protocolos[j];
						16:stCamara[i].config.stProtocolos[16] := Protocolos[j];
						17:stCamara[i].config.stProtocolos[17] := Protocolos[j];
						18:stCamara[i].config.stProtocolos[18] := Protocolos[j];
						19:stCamara[i].config.stProtocolos[19] := Protocolos[j];
						20:stCamara[i].config.stProtocolos[20] := Protocolos[j];
						21:stCamara[i].config.stProtocolos[21] := Protocolos[j];
						22:stCamara[i].config.stProtocolos[22] := Protocolos[j];
						23:stCamara[i].config.stProtocolos[23] := Protocolos[j];
						24:stCamara[i].config.stProtocolos[24] := Protocolos[j];
						25:stCamara[i].config.stProtocolos[25] := Protocolos[j];
						26:stCamara[i].config.stProtocolos[26] := Protocolos[j];
						27:stCamara[i].config.stProtocolos[27] := Protocolos[j];
						28:stCamara[i].config.stProtocolos[28] := Protocolos[j];
						29:stCamara[i].config.stProtocolos[29] := Protocolos[j];
						30:stCamara[i].config.stProtocolos[30] := Protocolos[j];
					END_CASE
				END_FOR
			END_FOR
			
			
			(*
			//Corre por todos os protocolos
			FOR i := DINT_TO_INT(uiBaixoArray) TO DINT_TO_INT(uiCimaArray) DO
				//apesar de o nome ser valvula ali em baixo é as camaras que vao receber esse protocolo
				F_StringSeparadorFBGrupos(sStr:= Protocolos[i].DB.Valvulas, ListaINT:=iValvulas);
				FOR j := 0 TO 500 DO
					IF iValvulas[j] = 0 THEN
						EXIT;
					END_IF
					
					IF iValvulas[j] < uiCimaArray + 1 THEN
						//encontra uma posição vazia no role
						FOR k := 0 TO 4 DO
							CASE k OF
								0:IF stCamara[iValvulas[j]].stProtocolos[0].DB.Nome = '' THEN EXIT; END_IF
								1:IF stCamara[iValvulas[j]].stProtocolos[1].DB.Nome = '' THEN EXIT; END_IF
								2:IF stCamara[iValvulas[j]].stProtocolos[2].DB.Nome = '' THEN EXIT; END_IF
								3:IF stCamara[iValvulas[j]].stProtocolos[3].DB.Nome = '' THEN EXIT; END_IF
								4:IF stCamara[iValvulas[j]].stProtocolos[4].DB.Nome = '' THEN EXIT; END_IF
							END_CASE
						END_FOR
						//se for > 4 siginifica que ja ocupou todas as posiçoes
						IF k < 4 THEN
							//joga o protocolo na posiçao vazia e o nome na posiçao vazia
							CASE k OF
								0:stCamara[iValvulas[j]].stProtocolos[0] := Protocolos[i];
								1:stCamara[iValvulas[j]].stProtocolos[1] := Protocolos[i];
								2:stCamara[iValvulas[j]].stProtocolos[2] := Protocolos[i];
								3:stCamara[iValvulas[j]].stProtocolos[3] := Protocolos[i];
								4:stCamara[iValvulas[j]].stProtocolos[4] := Protocolos[i];
							END_CASE
						END_IF
					END_IF
				END_FOR
			END_FOR
			*)
			
		END_IF
		
		iEstado := 2;
		xOcupado := false;
		
		2://fica esperando se muda algum deles
		
		IF xLeDoBanco THEN
			iEstado := 0;
		END_IF
		
		
		FOR i := DINT_TO_INT(uiBaixoArray) TO DINT_TO_INT(uiCimaArray) DO
			IF Protocolos[i].xEditado THEN
				iEstado := 3;
				iProtocoloAlterado := i;
				EXIT;
			END_IF
		END_FOR
		
		
		
		3:
		
			fbSB.Clear()
				.Append('UPDATE `geral`.`protocolo` SET `Nome` = $'')
				.Append(Protocolos[iProtocoloAlterado].DB.Nome)
				.Append('$', `NomeIHM` = $'')
				.Append(Protocolos[iProtocoloAlterado].DB.NomeIHM);
				
			sAux[0] := fbSB.GetString();
				
			fbSB.Clear()	
				.Append('$', `Valvulas` = $'')
				.Append(Protocolos[iProtocoloAlterado].DB.Valvulas);
				
			sAux[1] := fbSB.GetString();
			
			
			fbSB.Clear()
				.Append('$', `ET01TON` = $'')
				.Append(LREAL_TO_STRING(Protocolos[iProtocoloAlterado].DB.ET01TON))
				.Append('$', `ET01TOFF` = $'')
				.Append(LREAL_TO_STRING(Protocolos[iProtocoloAlterado].DB.ET01TOFF))
				.Append('$', `ET01NC` = $'')
				.Append(DINT_TO_STRING(Protocolos[iProtocoloAlterado].DB.ET01NC));
			
			sAux[2] := fbSB.GetString();
				
			fbSB.Clear()	
				.Append('$', `ET02TON` = $'')
				.Append(LREAL_TO_STRING(Protocolos[iProtocoloAlterado].DB.ET02TON))
				.Append('$', `ET02TOFF` = $'')
				.Append(LREAL_TO_STRING(Protocolos[iProtocoloAlterado].DB.ET02TOFF))
				.Append('$', `ET02NC` = $'')
				.Append(DINT_TO_STRING(Protocolos[iProtocoloAlterado].DB.ET02NC));
				
			sAux[3] := fbSB.GetString();
			
			fbSB.Clear()
				.Append('$', `ET03TON` = $'')
				.Append(LREAL_TO_STRING(Protocolos[iProtocoloAlterado].DB.ET03TON))
				.Append('$', `ET03TOFF` = $'')
				.Append(LREAL_TO_STRING(Protocolos[iProtocoloAlterado].DB.ET03TOFF))
				.Append('$', `ET03NC` = $'')
				.Append(DINT_TO_STRING(Protocolos[iProtocoloAlterado].DB.ET03NC));
				
			sAux[4] := fbSB.GetString();
				
			fbSB.Clear()
				.Append('$', `ET04TON` = $'')
				.Append(LREAL_TO_STRING(Protocolos[iProtocoloAlterado].DB.ET04TON))
				.Append('$', `ET04TOFF` = $'')
				.Append(LREAL_TO_STRING(Protocolos[iProtocoloAlterado].DB.ET04TOFF))
				.Append('$', `ET04NC` = $'')
				.Append(DINT_TO_STRING(Protocolos[iProtocoloAlterado].DB.ET04NC));
				
			sAux[5] := fbSB.GetString();
			
			fbSB.Clear()
				.Append('$', `ET05TON` = $'')
				.Append(LREAL_TO_STRING(Protocolos[iProtocoloAlterado].DB.ET05TON))
				.Append('$', `ET05TOFF` = $'')
				.Append(LREAL_TO_STRING(Protocolos[iProtocoloAlterado].DB.ET05TOFF))
				.Append('$', `ET05NC` = $'')
				.Append(DINT_TO_STRING(Protocolos[iProtocoloAlterado].DB.ET05NC));
			
			sAux[6] := fbSB.GetString();
				
			fbSB.Clear()
				.Append('$', `ET06TON` = $'')
				.Append(LREAL_TO_STRING(Protocolos[iProtocoloAlterado].DB.ET06TON))
				.Append('$', `ET06TOFF` = $'')
				.Append(LREAL_TO_STRING(Protocolos[iProtocoloAlterado].DB.ET06TOFF))
				.Append('$', `ET06NC` = $'')
				.Append(DINT_TO_STRING(Protocolos[iProtocoloAlterado].DB.ET06NC));
				
			sAux[7] := fbSB.GetString();
			
			fbSB.Clear()
				.Append('$', `ET07TON` = $'')
				.Append(LREAL_TO_STRING(Protocolos[iProtocoloAlterado].DB.ET07TON))
				.Append('$', `ET07TOFF` = $'')
				.Append(LREAL_TO_STRING(Protocolos[iProtocoloAlterado].DB.ET07TOFF))
				.Append('$', `ET07NC` = $'')
				.Append(DINT_TO_STRING(Protocolos[iProtocoloAlterado].DB.ET07NC));
			
			sAux[8] := fbSB.GetString();	
				
			fbSB.Clear()
				.Append('$', `ET08TON` = $'')
				.Append(LREAL_TO_STRING(Protocolos[iProtocoloAlterado].DB.ET08TON))
				.Append('$', `ET08TOFF` = $'')
				.Append(LREAL_TO_STRING(Protocolos[iProtocoloAlterado].DB.ET08TOFF))
				.Append('$', `ET08NC` = $'')
				.Append(DINT_TO_STRING(Protocolos[iProtocoloAlterado].DB.ET08NC));
				
			sAux[9] := fbSB.GetString();
			
			fbSB.Clear()
				.Append('$', `ET09TON` = $'')
				.Append(LREAL_TO_STRING(Protocolos[iProtocoloAlterado].DB.ET09TON))
				.Append('$', `ET09TOFF` = $'')
				.Append(LREAL_TO_STRING(Protocolos[iProtocoloAlterado].DB.ET09TOFF))
				.Append('$', `ET09NC` = $'')
				.Append(DINT_TO_STRING(Protocolos[iProtocoloAlterado].DB.ET09NC));
				
			sAux[10] := fbSB.GetString();
				
			fbSB.Clear()
				.Append('$', `ET10TON` = $'')
				.Append(LREAL_TO_STRING(Protocolos[iProtocoloAlterado].DB.ET10TON))
				.Append('$', `ET10TOFF` = $'')
				.Append(LREAL_TO_STRING(Protocolos[iProtocoloAlterado].DB.ET10TOFF))
				.Append('$', `ET10NC` = $'')
				.Append(DINT_TO_STRING(Protocolos[iProtocoloAlterado].DB.ET10NC))
				.Append('$', `xFinalDeSemana` = $'')
				.Append(DINT_TO_STRING(Protocolos[iProtocoloAlterado].DB.xFinalDeSemana));
				
			sAux[11] := fbSB.GetString();
			(*	*)
				
			fbSB.Clear()
				.Append('$' WHERE (`ID` = $'')
				.Append(DINT_TO_STRING(Protocolos[iProtocoloAlterado].DB.ID))
				.Append('$');');
			
			sAux[12] := fbSB.GetString();
			
			
			
			sCmdUpdate := F_ConcatArray1000(sAux);
			
			aPara.eParaType := E_ExpParameterType.STRING_;
			aPara.nParaSize := SIZEOF(sAux[0]);
			
			IF fbPLCDBCmd.Execute(
				hDBID:= 1, 
				pExpression:= ADR(sCmdUpdate), 
				cbExpression:= SIZEOF(sCmdUpdate), 
				pData:= ADR(sAuxVazio), 
				cbData:= SIZEOF(sAuxVazio), 
				pParameter:= ADR(aPara), 
				cbParameter:= SIZEOF(aPara))
			THEN
				Protocolos[iProtocoloAlterado].xEditado := FALSE;
				iEstado := 0;
				xLeDoBanco := TRUE;
				
				FOR i := DINT_TO_INT(uiBaixoArray) TO DINT_TO_INT(uiCimaArray) DO
					sNomeProtocoloIHM[i] := CONCAT(DINT_TO_STRING(Protocolos[i].DB.ID),CONCAT(' - ',Protocolos[i].DB.Nome));
				END_FOR
			END_IF
		
		
	END_CASE


ELSE
	
	ValidaLicensa();
END_IF

END_FUNCTION_BLOCK

// POUs/Automatico/Aspercao/ControleValvulas/BancoValvula/FB_IniciaValvulaBanco
FUNCTION_BLOCK FB_IniciaValvulaBanco
VAR_IN_OUT
	Valvulas : ARRAY[*] OF st_Valvula;
	ControleValvulas : ARRAY[*] OF st_ControleValvula;
END_VAR
VAR_INPUT
	xLe : BOOL;
END_VAR
VAR_OUTPUT
	xOcupado : BOOL;
END_VAR
VAR
	iEstado : INT;
	saAux : ARRAY[0..1000] OF STRING(80);
	stBanco : ARRAY[0..1000] OF st_BancoValvula;
	
	fbDBPuxa : FB_PLCDBCmdEvt(sNetID := '', tTimeout := T#10S);
    sCmd          : STRING (1000); 
    stPara         : ST_ExpParameter;
	sAux		  : STRING;
	
	diBaixo : DINT;
	diCima : DINT;
	diResultados : DINT;
	TagAProcurar		: STRING(80);
	
	i : INT;
	
	fbPLCDBCmd			: FB_PLCDBCmdEvt(sNetID := '', tTimeout := T#60S);
	fbSQLDatabase		: FB_SQLDatabaseEvt(sNetID := '', tTimeout := T#60S);
END_VAR




CASE iEstado OF 
	
	0 ://Esperando iniciar
	
		IF xLe THEN
			iEstado := 1;
			diBaixo := LOWER_BOUND(Valvulas,1);
			diCima := UPPER_BOUND(Valvulas,1);
		END_IF
	
	1: //abre conexao
			IF fbSqlDatabase.Connect(INT_TO_UDINT(1)) THEN
				IF fbSqlDatabase.bError THEN
					IF fbSqlDatabase.ipTcResult.ipSourceInfo.sName = 'ADSERR_DEVICE_LICENSENOTFOUND' THEN
						// se der isso ele nao fica tentando e gerando uma caralhada de erro pq nao tem a lisença
						iEstado := 0;
						xLe := false;
					ELSE
						iEstado := 2;
					END_IF
				ELSE
					IF fbSqlDatabase.bConnected THEN
						iEstado := 3;
					END_IF
				END_IF
			END_IF
	
		3: // le o role
			TagAProcurar		:= '';
			stPara.eParaType	:= E_ExpParameterType.STRING_;
			stPara.nParaSize	:= SIZEOF(TagAProcurar);
			stPara.sParaName	:= 'Tag';
	
			// set command with placeholder
			sCmd := CONCAT(CONCAT('SELECT * FROM ','geral.configvalvulas'),';');
	
			// call functionblock
			IF fbPLCDBCmd.ExecuteDataReturn
				(
					hDBID := 1,
						pExpression := ADR(sCmd),
						cbExpression := SIZEOF(sCmd),
						pData := ADR(TagAProcurar),
						cbData := SIZEOF(TagAProcurar),
						pParameter := ADR(stPara),
						cbParameter := SIZEOF(stPara),
						nStartIndex := 0,
						nRecordCount := DINT_TO_UDINT(diCima),
						pReturnData := ADR(stBanco),
						cbReturnData := SIZEOF(stBanco),
						pRecords := ADR(diResultados))
			THEN
				IF fbPLCDBCmd.bError THEN
					iEstado			:= 0;
					xLe := FALSE;
				ELSE
					
					iEstado	:= 4;
					xLe 	:= FALSE;
					FOR i := 1 TO TO_INT(diCima) DO
						Valvulas[i].en.sNome_Funcao := CONCAT(CONCAT(CONCAT('VS',TO_STRING(i)),' - '),stBanco[i-1].sNome);
						ControleValvulas[i].Config.sNomeValvulaIHM := stBanco[i-1].sNome;
					END_FOR
					
				END_IF
			END_IF
	
		4: // FechaConexao conexao
			IF fbSqlDatabase.Disconnect() THEN
	
	
				IF fbSqlDatabase.bError THEN
					iEstado := 0;
				ELSE
					iEstado := 0;
				END_IF
			END_IF
	
	
END_CASE

END_FUNCTION_BLOCK

// POUs/Automatico/Aspercao/ControleValvulas/FB_ControleValvulaApersao
FUNCTION_BLOCK FB_ControleValvulaApersao
VAR_IN_OUT
	stControle : st_ControleValvula;
END_VAR
VAR_INPUT	
	GUID			: STRING;//GUID do processo que vai ser feito na valvula, se for 0 é pq nao tem proceso rolando, ai nao pode aspergir
	xCamaraTempOK	: BOOL; //Temperatura da camera esta OK
	xCamaraUmidOK	: BOOL; //Umidade da camera esta OK
	xAnelPressOK	: BOOL; //Pressao do anel esta OK
	xTanqueTempOK	: BOOL; //Temperatura do tanque esta OK
	rTempAgua		: REAL; //temperatura da agua para o log no banco
	rPressaoAnel	: REAL;	//pressao da anel para o log no banco
	tsHoraAtual		: TIMESTRUCT; //Hora atual
	xCancela		: BOOL; //sinal de cancela o protocolo atual
	xPausaSincCluster : BOOL;//pausa para o sincronismo das valvulas do cluster
	xPausaSincEntreCluster : BOOL;//pausa para o sincronismo entre clusters
	xPausaSincCamaras : BOOL;//pausa para o sincronismo entre as camaras
END_VAR
VAR_OUTPUT
	iStatus 		: INT;
	xEmProcesso 	: BOOL;// se a valvula ja escolheu o protocolo e vai tentar aspergir
	sStatus 		: STRING;
	xPausado		: BOOL;
	sEtapaAtual		: STRING;
	tRestanteEtapa	: TIME; //Tempo ate terminar a etapa atual
	xLigaValvula	: BOOL;//Sinal interno mandando ligar a valvula
	iCicloAtual 	: INT; // qual o Ciclo que eles esta de todo protocolo
	dtHoraTermina 	: DT;// que hrs termina o protocolo
	sHoraTermina 	: STRING;//que hrs termina o protocolo
	xTempoMaximo	: BOOL;// se deu o tempo maximo de aspersao
	iTotalDeCiclos : INT;// quantidade de ciclos que o protocolo tem
	rEtapasSemMudar: ARRAY[1..10,1..3] OF LREAL;//etapas do processo
	iEtapaAtual : INT;//Etapa atual do processo
	xVSAr : BOOL;
END_VAR
VAR
	iEstado : INT;
	iEstadoBanco : INT;
	i : INT;
	k : INT;
	
	rEtapas 	: ARRAY[1..10,1..3] OF LREAL;
	iUltimaEtapa: INT;
	
	tonpEtapa	: TON_P;
	tEtapa		: TIME;
	
	stProtocoloSelecionado : st_Protocolo;
	stControleAnterior : st_ControleValvula;
	
	tsInicioCiclo	: TIMESTRUCT;
	tsFimCiclo		: TIMESTRUCT;
	
	dtAspergindo		: DT;
	dtNaoAspergindo		: DT;
	dtPausado			: DT;
	dtPausaUsuario		: DT;
	
	tAux				: ARRAY[0..10] OF TIME; 
	
	//grava o status da valvula
	fbPLCDBWrite	: FB_PLCDBWriteEvt(sNetID := '', tTimeout := T#30S); //Bloco para gravar no banco de dados
	xGravaLogValvula: BOOL;
	EstruturaBanco : st_ValvulasBD;

	ColumnNamesGrava : ARRAY[0..15] OF STRING(50) := ['ID',
														'Valvula',
														'Processo',
														'protocolo',
														'Ciclo',
														'Inicio',
														'Fim',
														'Aspergindo',
														'NaoAspergindo',
														'Pausado',
														'PausaUsuario',
														'vazao',
														'TemperaturaAgua',
														'PressaoAnel',
														'Cancelado',
														'Timestamp'];
													
						
    fbPLCDBCmd,fbDBCmdAF    : FB_PLCDBCmdEvt(sNetID := '', tTimeout := T#5S);
    sCmd          : STRING (1000); 
    aPara         : ST_ExpParameter;
	sAux 		  : STRING;
	xteste : BOOL;
	
	rtPulou : R_TRIG;
	
	xAdicioneiValvula : BOOL;
	
	rtLigaManu : R_TRIG;
	ftLigaManu : F_TRIG;
	
	
	fbSalvaEvento : ARRAY[0..15] OF FB_SalvaEventoRelatorio;
	
	saAux : ARRAY[0..50] OF STRING(80);//para gerar os comandos
	
	tsHoraInicio : TIMESTRUCT;
	dtHoraInicio : DT;
	dtPausaTotal : DT;
	dtAux : DT;
	dtAux2 : DT;
	j : INT;
	
	xCalculaHoraFinal1Vez : BOOL;
	
	btONOFF : B_TRIG;
	xSalvaONOFF :BOOL;
	
 	tonValvulaAberta: TON;//isso é nojento mas ta foda aqui 
	
	rtCancelouValvula : r_trig;
	
	sGuidAnterior : STRING;
	rtMudouGuid : r_TRIG;
	
	rtAbriuValvula : R_TRIG;
	
	tonTempoAntesDaAspersao : ton;
	
	tonAntesDoAr : TON;
	tonArAberto : TON;
	xFechouAValulaPorCiclo : BOOL;
	rtFechouAValulaPorCiclo : R_TRIG;
	
	xValvulaAbriu : BOOL;
	rtValvulaAbriu : R_TRIG;
	
	rtLigaManuAr : R_TRIG;
	ftLigaManuAr : F_TRIG;
	
	rtLigaBotao : R_TRIG;
	ton10s : TON;
	x10s : BOOL;
	ton5s : TON;
	x5s : BOOL;
	ton2s : TON;
	x2s : BOOL;
	ton500ms : TON;
	x500ms : BOOL;
	
	tonBTCancela : TON;
	xCancelaInterno : BOOL;
	rtCancelaInterno : R_TRIG;
	
	tonPausaBT : TON;
	xPausaBT : BOOL;
	rtPausaBT : R_TRIG;
	
END_VAR



(*
iStatus: 
	99: Esperando iniciar
	1: Pausado Sinc
	2: Pausado Critico
	3: Terrminou de aspergir
	4: Esperando
	5: Aspergindo
	6: Aspergindo Esperando
	7: Manual desligada
	8: Manual Ligada
	9: Cancelado
*)





IF xLicensaValida6446896834 THEN	

	AjustaEntrada();
	AjustaSaida();
	
	LogBanco();
	CancelaProtocolo();
	TempoMaximoDeProtocolo();
	EventosRelatorio();
	SalvaAbreEFecha();
	ControleEventos();
	VSAr();
	BotaoELed();
	
	
	stControle.EN.iIndexValvula := stControle.EN.stValvula.en.i;
	
	stControle.EN.stValvula.en.xEmergenciaOK := stControle.EN.xEmergenciaOK;
	
	
	rtMudouGuid(CLK:= GUID <> '', Q=> );
	IF rtMudouGuid.Q THEN
		IF GUID <> '' THEN
			sGuidAnterior := GUID;
		END_IF
	END_IF
	
	
	IF GUID = '' THEN
		stControle.sa.sTempoRestante := 'EspIni';
	ELSE
		dtAux := TIME_TO_DT(tRestanteEtapa);
		stControle.sa.sTempoRestante := REPLACE(STR1:= TO_STRING(dtAux), STR2:= '', L:= 15, P:=0);	
	END_IF
	
	//esse sinal garante que quando o controle dos cluster liberar o cluster dessa valvula ela vai ligar na hora, garantindo assim o sincronismo
	stControle.sa.xNaoLigoSoPorSincETC := xPausaSincEntreCluster AND xCamaraTempOK AND xCamaraUmidOK AND xAnelPressOK AND xTanqueTempOK OR xPausaBT OR stControle.EN.xPausaUsuarioCamara OR NOT stControle.EN.xEmergenciaOK AND NOT xPausaSincCluster AND NOT xPausaSincCamaras;
	stControle.sa.xPausadoSemSin := NOT xCamaraTempOK OR NOT xCamaraUmidOK OR NOT xAnelPressOK OR NOT xTanqueTempOK OR xPausaBT OR stControle.EN.xPausaUsuarioCamara OR NOT stControle.EN.xEmergenciaOK;
	
	
	//Tudo que pode pausar a valvula que nao é o numero max de valvulas
	IF (NOT xCamaraTempOK OR NOT xCamaraUmidOK OR NOT xAnelPressOK OR NOT xTanqueTempOK
		 OR xPausaSincCluster OR xPausaSincEntreCluster OR xPausaSincCamaras OR xPausaBT
		 OR stControle.EN.xPausaUsuarioCamara OR NOT stControle.EN.xEmergenciaOK) AND NOT xteste THEN
		xPausado := TRUE;
		
		//iStatus := 1; 	
		IF xPausaSincCluster THEN
			CASE stControle.Config.Linguagem OF
				enu_Linguagem.Portugues:	sStatus := ('Pausa para sincronizar com o cluster');
				enu_Linguagem.Espanhol: 	sStatus := ('Pausa para sincronizar con el clúster');
				enu_Linguagem.Ingles: 		sStatus := ('Pause to synchronize with the cluster');
			END_CASE
			stControle.sa.sTempoRestante := 'SinClus';
		END_IF
		IF xPausaSincEntreCluster THEN
			dtAux := TIME_TO_DT(stControle.EN.tTempoAteSinc);
			CASE stControle.Config.Linguagem OF
				enu_Linguagem.Portugues:	sStatus := CONCAT('Pausa para sincronizar entre os clusters por mais: ',REPLACE(STR1:= TO_STRING(dtAux), STR2:= '', L:= 15, P:=0));
				enu_Linguagem.Espanhol: 	sStatus := CONCAT('Pausa para sincronizar entre clusters para más: ',REPLACE(STR1:= TO_STRING(dtAux), STR2:= '', L:= 15, P:=0));
				enu_Linguagem.Ingles: 		sStatus := CONCAT('Pause to synchronize between clusters for more: ',REPLACE(STR1:= TO_STRING(dtAux), STR2:= '', L:= 15, P:=0));
			END_CASE
			stControle.sa.sTempoRestante := 'SinECL';
		END_IF
		IF xPausaSincCamaras THEN
			CASE stControle.Config.Linguagem OF
				enu_Linguagem.Portugues:	sStatus := 'Pausa para sincronizar entre as câmaras';
				enu_Linguagem.Espanhol: 	sStatus := 'Pausa para sincronizar entre cámaras';
				enu_Linguagem.Ingles: 		sStatus := 'Pause to synchronize between cameras';
			END_CASE
			stControle.sa.sTempoRestante := 'SinCAM';
		END_IF
		IF xPausaBT OR stControle.EN.xPausaUsuarioCamara THEN
			CASE stControle.Config.Linguagem OF
				enu_Linguagem.Portugues:	sStatus := ('Pausa do usuario');
				enu_Linguagem.Espanhol: 	sStatus := ('Pausa del user');
				enu_Linguagem.Ingles: 		sStatus := ('User$'s pause');
			END_CASE
			stControle.sa.sTempoRestante := 'PausaBT';
		END_IF	
		IF NOT xCamaraTempOK THEN
			CASE stControle.Config.Linguagem OF
				enu_Linguagem.Portugues:	sStatus := 'Temperatura da câmara fora de setpoint';
				enu_Linguagem.Espanhol: 	sStatus := 'Temperatura de la cámara fuera de consigna';
				enu_Linguagem.Ingles: 		sStatus := 'Chamber temperature out of setpoint';
			END_CASE
			stControle.sa.sTempoRestante := 'TempCam';
		END_IF
		IF NOT xCamaraUmidOK THEN
			CASE stControle.Config.Linguagem OF
				enu_Linguagem.Portugues:	sStatus := 'Umidade da câmara fora de setpoint';
				enu_Linguagem.Espanhol: 	sStatus := 'Humedad de cámara fuera de consigna';
				enu_Linguagem.Ingles: 		sStatus := 'Chamber humidity out of setpoint';
			END_CASE
			stControle.sa.sTempoRestante := 'UmiCam';
		END_IF
		IF NOT xAnelPressOK THEN
			CASE stControle.Config.Linguagem OF
				enu_Linguagem.Portugues:	sStatus := 'Pressão do anel abaixo de 0.5 Bar';
				enu_Linguagem.Espanhol: 	sStatus := 'Presión del anillo inferior a 0,5 Bar';
				enu_Linguagem.Ingles: 		sStatus := 'Ring pressure below 0.5 Bar';
			END_CASE
			stControle.sa.sTempoRestante := 'PreAnel';
		END_IF
		IF NOT xTanqueTempOK THEN
			CASE stControle.Config.Linguagem OF
				enu_Linguagem.Portugues:	sStatus := 'Temperatura do tanque acima de 4 ºC';
				enu_Linguagem.Espanhol: 	sStatus := 'Temperatura del depósito superior a 4 ºC';
				enu_Linguagem.Ingles: 		sStatus := 'Tank temperature above 4 ºC';
			END_CASE
			stControle.sa.sTempoRestante := 'TempRes';
		END_IF
		IF NOT stControle.EN.xEmergenciaOK THEN
			CASE stControle.Config.Linguagem OF
				enu_Linguagem.Portugues:	sStatus := 'Emergencia';
				enu_Linguagem.Espanhol: 	sStatus := 'Emergencia';
				enu_Linguagem.Ingles: 		sStatus := 'Emergency';
			END_CASE
			stControle.sa.sTempoRestante := 'EMER';
		END_IF
		
	ELSE
		xPausado := FALSE;
	END_IF
	
	//Seguranca caso fique sem guid por algum motivo, ai para de aspergir 
	IF GUID = '' THEN
		iEstado := 0;
		dtPausaTotal := DT#1970-01-01-00:00;
		tsHoraInicio := DT_TO_SYSTEMTIME(DT#1970-01-01-00:00);
		dtHoraTermina := (DT#1970-01-01-00:00);
		sHoraTermina := '';
		iEtapaAtual := 0;
		stControle.SA.xParaVentilacao := FALSE;
		xPausaSincCamaras := FALSE;
		xPausaSincEntreCluster := FALSE;
		xPausaSincCluster := FALSE;
		stControle.EN.xPausaUsuarioCamara := FALSE; 
	END_IF
	
	//So pode cancelar se tiver guid
	rtPulou(CLK:= GUID <> '' AND (stControle.EN.xPulaAspersao OR stControle.EN.xCancelaSupervisorio OR xCancelaInterno), Q=> );
	IF rtPulou.q THEN
		iEstado := 6;
		stControle.EN.xPulaAspersao := FALSE;
		xLigaValvula := FALSE;
		xCancelaInterno := false;
		
		//Se calcelou e tava aberto tem que tirar tb
		IF xAdicioneiValvula THEN
			stControle.EN.iValvulasAbertas := stControle.EN.iValvulasAbertas - 1;
			stControle.EN.iValvulasAbertasCamara := stControle.EN.iValvulasAbertasCamara -1;
			xAdicioneiValvula:= FALSE; 
		END_IF
	END_IF
	
	//bit so interno para jogar todas as valvulas para o fim da aspersao, pra caso a gente faça alteração no final de semana
	IF stControle.en.xFinalizaInterno THEN
		stControle.en.xFinalizaInterno := FALSE;
		iEstado := 4;
	END_IF
	
	
	
	CASE iEstado OF
		
		0: // Esperando processo iniciar
		
			stControle.SA.xParaVentilacao := FALSE;
			IF GUID <> '' THEN
				iEstado := 1;
			END_IF
			iStatus := 99;//Antes de inicar
			CASE stControle.Config.Linguagem OF
				enu_Linguagem.Portugues:	sStatus := 'Esperando processo iniciar';
				enu_Linguagem.Espanhol: 	sStatus := 'Esperando el inicio del proceso';
				enu_Linguagem.Ingles: 		sStatus := 'Waiting for process to start';
			END_CASE
			xLigaValvula := FALSE;
			iCicloAtual := 0;
			iTotalDeCiclos := 0;
			
			xEmProcesso := FALSE;
			
			
		1://Tem processo esperando a valvula selecionar o protocolo
		
			stControle.SA.xParaVentilacao := FALSE;
			
			IF stControle.EN.xLigaAutomaticoSupervisorio THEN
				stControle.EN.stProtocolos[0].xSelecionado := TRUE;
			END_IF
			
			FOR i := 0 TO 3 DO
				IF stControle.EN.stProtocolos[i].xSelecionado THEN
					
				
					dtHoraInicio := SYSTEMTIME_TO_DT(tsHoraAtual);
					
					IF stControle.EN.rTempoEsperaAntesAspergir = 0 THEN
						iEstado := 2;
					ELSE
						iEstado := 8;
						tonTempoAntesDaAspersao(IN:= FALSE);
					END_IF
					
					
					tsHoraInicio := tsHoraAtual;
					stControle.EN.stProtocolos[i].xSelecionado := FALSE;
					stProtocoloSelecionado := stControle.EN.stProtocolos[i];
					
					
					//joga em um array para ficar mais facil ali pra baixo
					rEtapas[1,1] := stProtocoloSelecionado.DB.ET01TON;
					rEtapas[1,2] := stProtocoloSelecionado.DB.ET01TOFF;
					rEtapas[1,3] := stProtocoloSelecionado.DB.ET01NC;
					rEtapas[2,1] := stProtocoloSelecionado.DB.ET02TON;
					rEtapas[2,2] := stProtocoloSelecionado.DB.ET02TOFF;
					rEtapas[2,3] := stProtocoloSelecionado.DB.ET02NC;
					rEtapas[3,1] := stProtocoloSelecionado.DB.ET03TON;
					rEtapas[3,2] := stProtocoloSelecionado.DB.ET03TOFF;
					rEtapas[3,3] := stProtocoloSelecionado.DB.ET03NC;
					rEtapas[4,1] := stProtocoloSelecionado.DB.ET04TON;
					rEtapas[4,2] := stProtocoloSelecionado.DB.ET04TOFF;
					rEtapas[4,3] := stProtocoloSelecionado.DB.ET04NC;
					rEtapas[5,1] := stProtocoloSelecionado.DB.ET05TON;
					rEtapas[5,2] := stProtocoloSelecionado.DB.ET05TOFF;
					rEtapas[5,3] := stProtocoloSelecionado.DB.ET05NC;
					rEtapas[6,1] := stProtocoloSelecionado.DB.ET06TON;
					rEtapas[6,2] := stProtocoloSelecionado.DB.ET06TOFF;
					rEtapas[6,3] := stProtocoloSelecionado.DB.ET06NC;
					rEtapas[7,1] := stProtocoloSelecionado.DB.ET07TON;
					rEtapas[7,2] := stProtocoloSelecionado.DB.ET07TOFF;
					rEtapas[7,3] := stProtocoloSelecionado.DB.ET07NC;
					rEtapas[8,1] := stProtocoloSelecionado.DB.ET08TON;
					rEtapas[8,2] := stProtocoloSelecionado.DB.ET08TOFF;
					rEtapas[8,3] := stProtocoloSelecionado.DB.ET08NC;
					rEtapas[9,1] := stProtocoloSelecionado.DB.ET09TON;
					rEtapas[9,2] := stProtocoloSelecionado.DB.ET09TOFF;
					rEtapas[9,3] := stProtocoloSelecionado.DB.ET09NC;
					rEtapas[10,1] := stProtocoloSelecionado.DB.ET10TON;
					rEtapas[10,2] := stProtocoloSelecionado.DB.ET10TOFF;
					rEtapas[10,3] := stProtocoloSelecionado.DB.ET10NC;
					
					rEtapasSemMudar := rEtapas;
					xCalculaHoraFinal1Vez := TRUE;
					HoraTermina();
					
					//Ve qual a ultima etapa
					IF 		stProtocoloSelecionado.DB.ET10NC <> 0 THEN
						iUltimaEtapa := 10;
					ELSIF 	stProtocoloSelecionado.DB.ET09NC <> 0 THEN
						iUltimaEtapa := 9;
					ELSIF 	stProtocoloSelecionado.DB.ET08NC <> 0 THEN
						iUltimaEtapa := 8;
					ELSIF 	stProtocoloSelecionado.DB.ET07NC <> 0 THEN
						iUltimaEtapa := 7;
					ELSIF 	stProtocoloSelecionado.DB.ET06NC <> 0 THEN
						iUltimaEtapa := 6;
					ELSIF 	stProtocoloSelecionado.DB.ET05NC <> 0 THEN
						iUltimaEtapa := 5;
					ELSIF 	stProtocoloSelecionado.DB.ET04NC <> 0 THEN
						iUltimaEtapa := 4;
					ELSIF 	stProtocoloSelecionado.DB.ET03NC <> 0 THEN
						iUltimaEtapa := 3;
					ELSIF 	stProtocoloSelecionado.DB.ET02NC <> 0 THEN
						iUltimaEtapa := 2;
					ELSE
						iUltimaEtapa := 1;
					END_IF
					
					EXIT;
				END_IF
			END_FOR
	
			dtAspergindo := DT#1970-01-01-00:00;
			dtNaoAspergindo := DT#1970-01-01-00:00;
			dtPausado := DT#1970-01-01-00:00;
			dtPausaTotal := DT#1970-01-01-00:00;
			
			
			iTotalDeCiclos := 0;
			FOR i := 1 TO 10 DO
				iTotalDeCiclos := iTotalDeCiclos + REAL_TO_INT(rEtapas[i,3]);
			END_FOR
			iCicloAtual := 0;
			
			
			iStatus := 4;//esperando
			stControle.sa.sTempoRestante := 'Aguarda';
			
			CASE stControle.Config.Linguagem OF
				enu_Linguagem.Portugues:	sStatus := 'Esperando selecionar protocolo';
				enu_Linguagem.Espanhol: 	sStatus := 'A la espera de seleccionar el protocolo';
				enu_Linguagem.Ingles: 		sStatus := 'Waiting to select the protocol';
			END_CASE
			xLigaValvula := FALSE;
			
			xEmProcesso := FALSE;
			
		8:// tem que contar um tempo antes
			
			stControle.sa.sTempoRestante := 'ContIni';
			
			CASE stControle.Config.Linguagem OF
				enu_Linguagem.Portugues:	sStatus := 'Contando tempo antes de iniciar';
				enu_Linguagem.Espanhol: 	sStatus := 'Contar el tiempo antes de empezar';
				enu_Linguagem.Ingles: 		sStatus := 'Counting time before starting';
			END_CASE
			iStatus := 1;//Pausado normal
			
			tonTempoAntesDaAspersao(IN:= TRUE, PT:= REAL_TO_TIME(stControle.EN.rTempoEsperaAntesAspergir * 1000 * 60), Q=> , ET=> );
			IF tonTempoAntesDaAspersao.q THEN
				tonTempoAntesDaAspersao(IN:= FALSE);
				iEstado := 2;
			END_IF
		
			
			
		2://Ajusta etapa
			FOR i := 1 TO 10 DO
				IF rEtapas[i,3] <> 0 THEN
					IF NOT xLigaValvula THEN
						tEtapa := LREAL_TO_TIME(rEtapas[i,1]*1000);
						xLigaValvula := TRUE;
						IF iCicloAtual <> 0 THEN // no primeiro ciclo tem o sincronismo que nao pode contar esse tempo
							tsInicioCiclo := tsHoraAtual;
						END_IF
					ELSE
						tEtapa := LREAL_TO_TIME(rEtapas[i,2]*1000*60);
						xLigaValvula := FALSE;
					END_IF
					iEtapaAtual := i;
					tonpEtapa(IN:= FALSE);	
					
					IF xLigaValvula AND tEtapa > T#1MS THEN// se tiver que abrir a valvula olha se da pra abrir ou se tem que esperar as outras termianrem
						IF stControle.EN.iValvulasAbertas >= stControle.EN.iMaxValvulas OR stControle.EN.iValvulasAbertasCamara >= stControle.EN.iMaxValvulasAbertasCamara THEN
							//Nao da pra abrir ainda entao vai pra outro estqado e fica esperando
							iEstado := 5;
						ELSE
							//Marca que tem mais uma aberta e parte pra asperçao
							iEstado := 3;
							stControle.EN.iValvulasAbertas := stControle.EN.iValvulasAbertas + 1;
							stControle.EN.iValvulasAbertasCamara := stControle.EN.iValvulasAbertasCamara + 1;
							xAdicioneiValvula := TRUE;
						END_IF
					ELSE
						iEstado := 3;
					END_IF
					
					EXIT;
				END_IF
				IF i > iUltimaEtapa THEN
					xGravaLogValvula := TRUE;
					tsFimCiclo := tsHoraAtual;
					iCicloAtual := iCicloAtual + 1;
					AjustaBanco();
					
					iEstado := 4;
					EXIT;
				END_IF
			END_FOR
			
			
			xEmProcesso := TRUE;
		
		
		3://executa
		
			//Parte do principio que esta pausado ou que deu pau em tudo, se tiver fazendo outra coisa ai ele mostra aqui
			IF (NOT xCamaraTempOK OR NOT xCamaraUmidOK OR NOT xAnelPressOK OR NOT xTanqueTempOK OR NOT stControle.EN.xEmergenciaOK) THEN
				iStatus := 2; // Falha sistema critico
			ELSE
				iStatus := 1; // Pausado
			END_IF
		
			
			tonpEtapa(
			IN:= TRUE, 
			PT:= tEtapa, 
			PAUSE:= xPausado,
			Q=> , 
			ET=> );
			
			tRestanteEtapa := tonpEtapa.PT - tonpEtapa.ET;
			
			
			IF NOT xPausado THEN
				IF xLigaValvula THEN
					IF tRestanteEtapa > T#1MS THEN
						
						CASE stControle.Config.Linguagem OF
							enu_Linguagem.Portugues:	sStatus := CONCAT('Válvula aberta por mais ',TIME_TO_STRING(tRestanteEtapa));
							enu_Linguagem.Espanhol: 	sStatus := CONCAT('Válvula abierta para más ',TIME_TO_STRING(tRestanteEtapa));
							enu_Linguagem.Ingles: 		sStatus := CONCAT('Valve open for more ',TIME_TO_STRING(tRestanteEtapa));
						END_CASE
						iStatus := 5;// aspergindo
					END_IF
					stControle.SA.xParaVentilacao := TRUE;
				ELSE
					
					CASE stControle.Config.Linguagem OF
						enu_Linguagem.Portugues:	sStatus := CONCAT('Válvula fechada por mais ',TIME_TO_STRING(tRestanteEtapa));
						enu_Linguagem.Espanhol: 	sStatus := CONCAT('Válvula cerrada para más ',TIME_TO_STRING(tRestanteEtapa));
						enu_Linguagem.Ingles: 		sStatus := CONCAT('Valve closed for more ',TIME_TO_STRING(tRestanteEtapa));
					END_CASE
					iStatus := 6;// esperando para aspergir
					//se o tempo de aspersao for maior que o que falta ou se o tempo que ja roudou do timer for menor que o tempo que tem que ficar pausado depois ele diz pra para a ventilação
					stControle.SA.xParaVentilacao := iTotalDeCiclos > iCicloAtual + 1 AND (tRestanteEtapa < INT_TO_TIME(stControle.EN.iSegDesligarVentilacao * 1000) OR tonpEtapa.ET < INT_TO_TIME(stControle.EN.iSegDesligarVentilacao * 1000));
				END_IF
			ELSE
				//Se pasou nao por sincronismo para tudo
				IF stControle.sa.xPausadoSemSin THEN
					stControle.SA.xParaVentilacao := FALSE;
				ELSE
					stControle.SA.xParaVentilacao := stControle.EN.tTempoAteSinc < INT_TO_TIME(stControle.EN.iSegDesligarVentilacao * 1000);
				END_IF
			END_IF
			
			IF tonpEtapa.Q THEN
				tEtapa := T#0S;
				iEstado := 2;
				//Se a valvula ta off é porque é o fim do ciclo
				IF NOT xLigaValvula THEN
					//Ajusta etapa
					rEtapas[iEtapaAtual,3] := rEtapas[iEtapaAtual,3] - 1;
					iEstadoBanco := 1;
					
					//manda o banco salvar
					xGravaLogValvula := TRUE;
					//Ajusta os valores para salvar
					tsFimCiclo := tsHoraAtual;
					iCicloAtual := iCicloAtual + 1;
					AjustaBanco();
					//zera os valores pro proximo ciclo
					dtAspergindo := DT#1970-01-01-00:00;
					dtNaoAspergindo := DT#1970-01-01-00:00;
					dtPausado := DT#1970-01-01-00:00;
					dtPausaUsuario := DT#1970-01-01-00:00;
				ELSE
					IF xAdicioneiValvula THEN
						//Se a valvula ta ligada e acabou o temop ela vai fechar entao pode liberar para o proxima valvula comçar
						stControle.EN.iValvulasAbertas := stControle.EN.iValvulasAbertas - 1;
						stControle.EN.iValvulasAbertasCamara := stControle.EN.iValvulasAbertasCamara - 1;
						xAdicioneiValvula := FALSE;
					END_IF
				END_IF
			END_IF	
		
			//Esse cancelado vai voltar para o inicio nao ta sendo usado
			IF xCancela THEN
				//Volta pro estado 1 pq tem que escolher de novo o protocolo
				iEstado := 1;
				xLigaValvula := FALSE;
				stControle.sa.sTempoRestante := 'Cancel';
				//o proprio xCancela ja da true na parte do banco e cancela o que rolou aqui
				
				//Se calcelou e tava aberto tem que tirar tb
				IF xAdicioneiValvula THEN
					stControle.EN.iValvulasAbertas := stControle.EN.iValvulasAbertas - 1;
					stControle.EN.iValvulasAbertasCamara := stControle.EN.iValvulasAbertasCamara - 1;
					xAdicioneiValvula := FALSE;
				END_IF
			END_IF
			
			
			//se deu o tempo maximo de aspersao vai para outro estado que considera finalizado mas salva no banco que deu tempo max
			IF xTempoMaximo THEN
				iEstado := 7;
			END_IF
			
			
			xEmProcesso := TRUE;
		
		4://Terminou a asperção fica esperando reiniciar o processo
		
			stControle.SA.xFinalizou := TRUE;
			xLigaValvula := FALSE;
			stControle.sa.sTempoRestante := 'Fim';
			stControle.SA.xParaVentilacao := FALSE;
			
			CASE stControle.Config.Linguagem OF
				enu_Linguagem.Portugues:	sStatus := 'Terminou asperção';
				enu_Linguagem.Espanhol: 	sStatus := 'Aspersión finalizada';
				enu_Linguagem.Ingles: 		sStatus := 'Sprinkling finished';
			END_CASE
			iStatus := 3;//terminou de aspergir
			//Terminou o processo da camara ele tira o guid e volta pro inicio
			IF GUID = '' THEN
				//Caso o operador tenha clicado para iniciar de novo e nao era pra iniciar de novo
				stControle.EN.stProtocolos[0].xSelecionado := FALSE;
				stControle.EN.stProtocolos[1].xSelecionado := FALSE;
				stControle.EN.stProtocolos[2].xSelecionado := FALSE;
				stControle.EN.stProtocolos[3].xSelecionado := FALSE;
				iEstado := 0;
				stControle.SA.xFinalizou := FALSE;
			END_IF
			
			xEmProcesso := TRUE;
			
